# B&R Automation Studio project NewPendant_NG4_11_05_25A (part 10)

### HeadConfig.c
```c
/********************************************************************
 * COPYRIGHT --
 ********************************************************************
 * Package: FourAxisTigCtrl
 * File: HeadConfig.c
 * Author: ckaczkowski
 * Created: April 27, 2015
 * Directions - implemented 7 Febr 2018
   	TML_MTR_INST[i]._cfg.rev_motor - negative value change direction in Vel , Torq and Volt mode
	TML_MTR_INST[i]._cfg.rev_scale - negative value change pos and vel feedback (NOT Movement direction) and move direction in PT mode
 *******************************************************************/

#include <bur/plctypes.h>
#ifdef _DEFAULT_INCLUDES
	#include <AsDefault.h>
#endif

#include <math.h>

#ifndef _HEADCONFIG_C
#define _HEADCONFIG_C

#include <..\GlobDef.h>
#include <..\GlobDecl.h>
#include <..\..\Lib\LCDLib.c>

DINT NextDivider(DINT *in , DINT mod , BOOL dir);
DINT PickPinsNo(DINT *indx , DINT mod  );
void ParametrAssignToPointers(MASTER_typ *m  , UINT indx);

DINT ConfigureHead(MASTER_typ *m  , UINT headType );

DINT Configure_U_BEND_HP_PINS(MASTER_typ *m  , UINT headType );
DINT Configure_U_BEND_HP_ENC(MASTER_typ * m,UINT headType);
DINT Configure_OMEGA_16INCH_HP_ENCODER(MASTER_typ *m  , UINT headType );
DINT Configure_BPV_FACE_OSC(MASTER_typ * m, UINT headType);
DINT Configure_SUPER_MINI(MASTER_typ * m, UINT headType);
DINT Configure_U_BEND_HP_ENC_BEMF(MASTER_typ * m,UINT headType);
DINT Configure_BPV_F_HEAD(MASTER_typ * m, UINT headType);
DINT Configure_F_HEAD_HP_ENCODER(MASTER_typ * m,UINT headType);
DINT Configure_F_HEAD_HP_ENC_BEMF(MASTER_typ * m , UINT headType);
DINT Configure_BPV_FACE_OSC_ENC(MASTER_typ * m, UINT headType);
DINT Configure_BPV_FACE_OSC_EXP(MASTER_typ * m, UINT headType);
DINT Configure_BPV2_FACE_OSC_EXP(MASTER_typ * m, UINT headType);

DINT Configure_M_94(MASTER_typ * m, UINT headType);
DINT Configure_BPV_v2(MASTER_typ * m, UINT headType);
DINT Configure_MIG_TIG(MASTER_typ * m, UINT headType);

DINT Configure_BPV_v2_MPBO(MASTER_typ * m, UINT headType);
DINT Configure_BPV_v2_MPGH(MASTER_typ * m, UINT headType);
DINT Configure_BPV_v2_MPGV(MASTER_typ * m, UINT headType);

DINT Configure_BPV_v2_TT_BO(MASTER_typ * m, UINT headType);
DINT Configure_BPV_v2_MT_BO(MASTER_typ * m, UINT headType);

DINT Configure_BPV_v2_MT_BO_TOS(MASTER_typ * m, UINT headType);
DINT Configure_BPV_v2_TT_BO_TOS(MASTER_typ * m, UINT headType);

DINT  Configure_F_HEAD_HP_MINI_ENC(MASTER_typ * m,UINT headType);

DINT Configure_RUBIX(MASTER_typ * m, UINT headType);
DINT Configure_F_HEAD_MINI_STND(MASTER_typ * m,UINT headType);
DINT Configure_F_HEAD_MINI_OMEGA(MASTER_typ * m,UINT headType);
DINT Configure_D_HEAD_HP(MASTER_typ * m,UINT headType);

DINT Configure_CLAMSHELL_HEAD(MASTER_typ * m, UINT headType);
DINT Configure_CHERRYPOINT_BPV1_HEAD(MASTER_typ * m, UINT headType);
DINT Configure_CHERRYPOINT_BPV2_HEAD(MASTER_typ * m, UINT headType);
DINT Configure_CHERRYPOINT_MT_BP2_HEAD(MASTER_typ * m, UINT headType);

DINT  DefaultCalibr_U_BEND_HP_PINS(CurCalib_typ* defCalib);
DINT  DefaultCalibr_OMEGA_16INCH_HP_ENCODER(CurCalib_typ* defCalib);
DINT  DefaultCalibr_F_HEAD_HP_ENCODER(CurCalib_typ* defCalib);
DINT  DefaultCalibr_BPV_F_HEAD(CurCalib_typ* defCalib);

DINT Configure_BPV_v2_MT(MASTER_typ * m, UINT headType);
DINT Configure_BPV_V1_MT(MASTER_typ * m, UINT headType);

DINT  DefaultCalibr_F_HEAD_HP_MINI_ENC(CurCalib_typ* defCalib);
DINT  DefaultCalibr_U_BEND_HP_ENC(CurCalib_typ* defCalib);
DINT  DefaultCalibr_BPV_FACE_OSC(CurCalib_typ* defCalib);
DINT  DefaultCalibr_SUPER_MINI(CurCalib_typ* defCalib);
DINT  DefaultCalibr_U_BEND_HP_ENC_BEMF(CurCalib_typ* defCalib);
DINT  DefaultCalibr_F_HEAD_HP_ENC_BEMF(CurCalib_typ* defCalib);
DINT  DefaultCalibr_M_94(CurCalib_typ* defCalib);
DINT  DefaultCalibr_BPV_v2(CurCalib_typ* defCalib);
DINT  DefaultCalibr_BPV_v2_MPBO(CurCalib_typ* defCalib);
DINT  DefaultCalibr_BPV_v2_MPGH(CurCalib_typ* defCalib);
DINT  DefaultCalibr_BPV_v2_MPGV(CurCalib_typ* defCalib);

DINT  DefaultCalibr_BPV_v2_TT_BO(CurCalib_typ* defCalib);
DINT  DefaultCalibr_BPV_v2_MT_BO(CurCalib_typ* defCalib);

DINT  DefaultCalibr_BPV_v2_MT_BO_TOS(CurCalib_typ* defCalib);
DINT  DefaultCalibr_BPV_v2_TT_BO_TOS(CurCalib_typ* defCalib);

DINT  DefaultCalibr_RUBIX(CurCalib_typ* defCalib);
DINT  DefaultCalibr_F_HEAD_MINI_STND(CurCalib_typ* defCalib);
DINT  DefaultCalibr_F_HEAD_MINI_OMEGA(CurCalib_typ* defCalib);
DINT  DefaultCalibr_D_HEAD_HP(CurCalib_typ* defCalib);

DINT  DefaultCalibr_BPV_v2_MT(CurCalib_typ* defCalib);
DINT  DefaultCalibr_BPV_V1_MT(CurCalib_typ* defCalib);

DINT  DefaultCalibr_CLAMSHELL_HEAD(CurCalib_typ* defCalib);
DINT  DefaultCalibr_CHERRYPOINT_BPV1_HEAD(CurCalib_typ* defCalib);
DINT  DefaultCalibr_CHERRYPOINT_BPV2_HEAD(CurCalib_typ* defCalib);
DINT  DefaultCalibr_MIG_TIG(CurCalib_typ* defCalib);

float Gen_one;

DINT ConfigureHead(MASTER_typ *m  , UINT headType ){
int i;

CurCfg_typ *curCfg;
Cfg_typ *cfg;
CurCalib_typ *curCalib , *defaultCalib;

	if(!m)
		return;

	curCfg = (CurCfg_typ*)m->pCurCfg;
	cfg = (Cfg_typ*)m->pCfg;

	curCalib = m->pCalib;
	defaultCalib = m->pDefaultCalib;

	if(!curCfg || !cfg || !curCalib  || !defaultCalib)
		return;

	///
	if(curCalib->GenSetup[SETUP_POLE_ELEMENTS] < 2)
		curCalib->GenSetup[SETUP_POLE_ELEMENTS] = 2;

	else if(curCalib->GenSetup[SETUP_POLE_ELEMENTS] > 32)
		curCalib->GenSetup[SETUP_POLE_ELEMENTS] = 32;
	/////////

	for(i = 0 ; i < PROCESS_NUM ; i++)
		Process[i].ConfigReady = 0;

	for(i = 0 ; i < TML_SERVO_NUM ; i++){
		TML_MTR_INST[i].pState = 0;
		TML_MTR_INST[i]._cfg.NotAutoDownload = 0; // Default - auto download setup
		TML_MTR_INST[i]._cfg.MtrType = 0; // Default - DC Motor
	}

	for(i=0 ; i < VECTORS_NUM; i++){

		VectorStateMach[i].Indx = i;
	}

	// This is only to not forget Synch Configuration
	WIRE_Param_Set[0].pSynchMode = &WFSynchMode;
	WIRE_Param_Set[0].pSynchClock = &SynchClckToWF;

	WIRE_Param_Set[1].pSynchMode = &WPSynchMode;
	WIRE_Param_Set[1].pSynchClock = &SynchClckToWP;

	TVL_ROT_Param_Set[0].pSynchMode = &TVLSynchMode;
	TVL_ROT_Param_Set[0].pSynchClock = &SynchClckToTVL;

	////////////   NEW HEAD Configuration - will be from file parser   /////////////////////
	switch(headType){
		/************ 0 **********/
		case U_BEND_HP_PINS:

			// TVL
			m->pCfg->HeadCfg.SwitchHead.VECT_Indx = 0;
			m->pCfg->HeadCfg.SwitchHead.TML_Indx = 0;

			m->pCfg->HeadCfg.TVL.PROC_Indx = PROC_TVL;
			m->pCfg->HeadCfg.TVL.TML_Indx = TML_AX_TVL;
			m->pCfg->HeadCfg.TVL.DC_Indx = 0;

			m->pCfg->HeadCfg.TVL.VECT_Indx = VECT_TVL;
			m->pCfg->HeadCfg.TVL.Enc_Dir = 1;
			m->pCfg->HeadCfg.TVL.EncPerTick = 160;
			m->pCfg->HeadCfg.TVL.PinsPerRot = 0;  // Dynamic Configuration
			m->pCfg->HeadCfg.TVL.DistPerTick = 25.4 / 4.0; // 1/4"

			// Lamp On Off
			m->pCfg->HeadCfg.LampOnOFF.VECT_A_Indx = 0; // 0 - not used
			m->pCfg->HeadCfg.LampOnOFF.VECT_B_Indx = 0; // 0 - not used

			// INDX
			m->pCfg->HeadCfg.INDX.PROC_Indx = PROC_INDX; // Must be even is disabled

			m->pCfg->HeadCfg.OSC.DwellDir = 1;

		break;

		/************ 1 ************/
		case U_BEND_HP_ENC:

			m->pCfg->HeadCfg.GEN.Torch_Mode = MODE_SINGLE_TORCH;

			// TVL
			m->pCfg->HeadCfg.SwitchHead.VECT_Indx = 0;
			m->pCfg->HeadCfg.SwitchHead.TML_Indx = 0;

			m->pCfg->HeadCfg.TVL.PROC_Indx = PROC_TVL;
			m->pCfg->HeadCfg.TVL.TML_Indx = TML_AX_TVL;
			m->pCfg->HeadCfg.TVL.DC_Indx = 0;

			m->pCfg->HeadCfg.TVL.VECT_Indx = VECT_TVL;
			m->pCfg->HeadCfg.TVL.Enc_Dir = 1;
			m->pCfg->HeadCfg.TVL.EncPerTick = 200; // (4000 * 4) / (10 * 1/4") * 32 ( becaue 1/32" is one tick")
			m->pCfg->HeadCfg.TVL.PinsPerRot = 640;  // 80 pins , 1/4" per pin
			m->pCfg->HeadCfg.TVL.DistPerTick = 25.4 /32.0; // 1/32"

			m->pCfg->HeadCfg.TVL.BtnJog_Gain = 24;
			m->pCfg->HeadCfg.TVL.BtnJog_Mode = BTN_JOG_MODE_SINGLE;

			// WF
			m->pCfg->HeadCfg.WF.PROC_Indx = PROC_WIRE_FEED;
			m->pCfg->HeadCfg.WF.VECT_A_Indx = VECT_WF;
			m->pCfg->HeadCfg.WF.VECT_B_Indx = VECT_WF_1;
			m->pCfg->HeadCfg.WF.DC_A_Indx = DC_AX_WF;
			m->pCfg->HeadCfg.WF.DC_B_Indx = DC_AX_WF_1;

			m->pCfg->HeadCfg.WF.BtnJog_Gain = 24;
			m->pCfg->HeadCfg.WF.BtnJog_Mode = BTN_JOG_MODE_SINGLE;

			// WP
			m->pCfg->HeadCfg.WP.PROC_Indx = PROC_WIRE_PULSE;
			m->pCfg->HeadCfg.WP.VECT_A_Indx = VECT_WP;
			m->pCfg->HeadCfg.WP.VECT_B_Indx = VECT_WP_1;
			m->pCfg->HeadCfg.WP.DC_A_Indx = DC_AX_WP;
			m->pCfg->HeadCfg.WP.DC_B_Indx = DC_AX_WP_1;

			// OSC
			m->pCfg->HeadCfg.OSC.PROC_Indx = PROC_OSC;
			m->pCfg->HeadCfg.OSC.VECT_A_Indx = VECT_OSC;
			m->pCfg->HeadCfg.OSC.VECT_B_Indx = VECT_OSC;
			m->pCfg->HeadCfg.OSC.TML_A_Indx = TML_AX_OSC;
			m->pCfg->HeadCfg.OSC.TML_B_Indx = TML_AX_OSC;
			m->pCfg->HeadCfg.OSC.Limits_Harcoded = 0;

			m->pCfg->HeadCfg.OSC.BtnJog_Gain = 24.0;
			m->pCfg->HeadCfg.OSC.BtnJog_Mode = BTN_JOG_MODE_SINGLE;

			m->pCfg->HeadCfg.OSC.WheelJog_Gain1 = 5;
			m->pCfg->HeadCfg.OSC.WhelJog_Mode1 = WHL_JOG_MODE_STEP;

			m->pCfg->HeadCfg.OSC.WheelJog_Gain2 = 0.2;
			m->pCfg->HeadCfg.OSC.WhelJog_Mode2 = WHL_JOG_MODE_STEP;
			m->pCfg->HeadCfg.OSC.WhelJog_OnlyWhenRun = 1;

			m->pCfg->HeadCfg.OSC.DwellDir = 1;

			// AVC
			m->pCfg->HeadCfg.AVC.PROC_Indx = PROC_AVC;
			m->pCfg->HeadCfg.AVC.VECT_A_Indx = VECT_AVC;
			m->pCfg->HeadCfg.AVC.VECT_B_Indx = VECT_AVC;
			m->pCfg->HeadCfg.AVC.TML_A_Indx = TML_AX_AVC;
			m->pCfg->HeadCfg.AVC.TML_B_Indx = TML_AX_AVC;

			m->pCfg->HeadCfg.AVC.BtnJog_Gain = 24;
			m->pCfg->HeadCfg.AVC.BtnJog_Mode = BTN_JOG_MODE_SINGLE;

			// GAS
			m->pCfg->HeadCfg.GAS.PROC_Indx = PROC_GAS;

			// COOL
			m->pCfg->HeadCfg.COOL.PROC_Indx = PROC_COOL;

			// TIG
			m->pCfg->HeadCfg.TIG.PROC_Indx = PROC_TIG_PS;

			// HW
			m->pCfg->HeadCfg.HW.PROC_Indx = PROC_HW_PS;

			// INDX
			m->pCfg->HeadCfg.INDX.PROC_Indx = PROC_INDX; // Must be even is disabled

			// WB
			m->pCfg->HeadCfg.WB[WB_UD].PROC_Indx = PROC_WB_UD;
			m->pCfg->HeadCfg.WB[WB_LR].PROC_Indx = PROC_WB_LR;

			m->pCfg->HeadCfg.WB[WB_UD].VECT_Indx = VECT_WB_UD;
			m->pCfg->HeadCfg.WB[WB_LR].VECT_Indx = VECT_WB_LR;

			// Lamp On Off
			m->pCfg->HeadCfg.LampOnOFF.VECT_A_Indx = 0; // 0 - not used
			m->pCfg->HeadCfg.LampOnOFF.VECT_B_Indx = 0; // 0 - not used

			// frame size if zero always speed factor is 1.0
			m->FrameDia = 4.5 * in_2_mm ;
			m->FrameDia = 0.0;

			Configure_U_BEND_HP_ENC(m , U_BEND_HP_ENC);
			DefaultCalibr_U_BEND_HP_ENC(m->pDefaultCalib);

		break;

		/************ 2 ************/
		case F_HEAD_HP_ENCODER:

			m->pCfg->HeadCfg.GEN.Torch_Mode = MODE_SINGLE_TORCH;

			// TVL
			m->pCfg->HeadCfg.SwitchHead.VECT_Indx = 0;
			m->pCfg->HeadCfg.SwitchHead.TML_Indx = 0;

			m->pCfg->HeadCfg.TVL.PROC_Indx = PROC_TVL;
			m->pCfg->HeadCfg.TVL.TML_Indx = TML_AX_TVL;
			m->pCfg->HeadCfg.TVL.DC_Indx = 0;

			m->pCfg->HeadCfg.TVL.VECT_Indx = VECT_TVL;
			m->pCfg->HeadCfg.TVL.Enc_Dir = 1;
			m->pCfg->HeadCfg.TVL.EncPerTick = 38;  // 1/16 inch
			m->pCfg->HeadCfg.TVL.PinsPerRot = 0;  // Dynamic Configuration
			m->pCfg->HeadCfg.TVL.DistPerTick = 25.4 /16.0; // 1/16"

			m->pCfg->HeadCfg.TVL.BtnJog_Gain = 24;
			m->pCfg->HeadCfg.TVL.BtnJog_Mode = BTN_JOG_MODE_SINGLE;

			// WF
			m->pCfg->HeadCfg.WF.PROC_Indx = PROC_WIRE_FEED;
			m->pCfg->HeadCfg.WF.VECT_A_Indx = VECT_WF;
			m->pCfg->HeadCfg.WF.VECT_B_Indx = VECT_WF_1;
			m->pCfg->HeadCfg.WF.DC_A_Indx = DC_AX_WF;
			m->pCfg->HeadCfg.WF.DC_B_Indx = DC_AX_WF_1;

			m->pCfg->HeadCfg.WF.BtnJog_Gain = 24;
			m->pCfg->HeadCfg.WF.BtnJog_Mode = BTN_JOG_MODE_SINGLE;

			// WP
			m->pCfg->HeadCfg.WP.PROC_Indx = PROC_WIRE_PULSE;
			m->pCfg->HeadCfg.WP.VECT_A_Indx = VECT_WP;
			m->pCfg->HeadCfg.WP.VECT_B_Indx = VECT_WP_1;
			m->pCfg->HeadCfg.WP.DC_A_Indx = DC_AX_WP;
			m->pCfg->HeadCfg.WP.DC_B_Indx = DC_AX_WP_1;

			// OSC
			m->pCfg->HeadCfg.OSC.PROC_Indx = PROC_OSC;
			m->pCfg->HeadCfg.OSC.VECT_A_Indx = VECT_OSC;
			m->pCfg->HeadCfg.OSC.VECT_B_Indx = VECT_OSC;
			m->pCfg->HeadCfg.OSC.TML_A_Indx = TML_AX_OSC;
			m->pCfg->HeadCfg.OSC.TML_B_Indx = TML_AX_OSC;
			m->pCfg->HeadCfg.OSC.Limits_Harcoded = 0;

			m->pCfg->HeadCfg.OSC.BtnJog_Gain = 24.0;
			m->pCfg->HeadCfg.OSC.BtnJog_Mode = BTN_JOG_MODE_SINGLE;

			m->pCfg->HeadCfg.OSC.WheelJog_Gain1 = 5.0;
			m->pCfg->HeadCfg.OSC.WhelJog_Mode1 = WHL_JOG_MODE_STEP;

			m->pCfg->HeadCfg.OSC.WheelJog_Gain2 = 0.2;
			m->pCfg->HeadCfg.OSC.WhelJog_Mode2 = WHL_JOG_MODE_STEP;
			m->pCfg->HeadCfg.OSC.WhelJog_OnlyWhenRun = 1;

			m->pCfg->HeadCfg.OSC.DwellDir = 1;

			// AVC
			m->pCfg->HeadCfg.AVC.PROC_Indx = PROC_AVC;
			m->pCfg->HeadCfg.AVC.VECT_A_Indx = VECT_AVC;
			m->pCfg->HeadCfg.AVC.VECT_B_Indx = VECT_AVC;
			m->pCfg->HeadCfg.AVC.TML_A_Indx = TML_AX_AVC;
			m->pCfg->HeadCfg.AVC.TML_B_Indx = TML_AX_AVC;

			m->pCfg->HeadCfg.AVC.BtnJog_Gain = 24;
			m->pCfg->HeadCfg.AVC.BtnJog_Mode = BTN_JOG_MODE_SINGLE;

			// GAS
			m->pCfg->HeadCfg.GAS.PROC_Indx = PROC_GAS;

			// COOL
			m->pCfg->HeadCfg.COOL.PROC_Indx = PROC_COOL;

			// TIG
			m->pCfg->HeadCfg.TIG.PROC_Indx = PROC_TIG_PS;

			// HW
			m->pCfg->HeadCfg.HW.PROC_Indx = PROC_HW_PS;

			// INDX
			m->pCfg->HeadCfg.INDX.PROC_Indx = PROC_INDX; // Must be even is disabled

			// WB
			m->pCfg->HeadCfg.WB[WB_UD].PROC_Indx = PROC_WB_UD;
			m->pCfg->HeadCfg.WB[WB_LR].PROC_Indx = PROC_WB_LR;

			m->pCfg->HeadCfg.WB[WB_UD].VECT_Indx = VECT_WB_UD;
			m->pCfg->HeadCfg.WB[WB_LR].VECT_Indx = VECT_WB_LR;

			// Lamp On Off
			m->pCfg->HeadCfg.LampOnOFF.VECT_A_Indx = 0; // 0 - not used
			m->pCfg->HeadCfg.LampOnOFF.VECT_B_Indx = 0; // 0 - not used

			/////////////////////////////////////////////////////

			// frame size if zero always speed factor is 1.0
			//m->FrameDia = 4.5 * in_2_mm ;
			m->FrameDia = 0.0;

			Configure_F_HEAD_HP_ENCODER(m , F_HEAD_HP_ENCODER);
			DefaultCalibr_F_HEAD_HP_ENCODER(m->pDefaultCalib);

		break;

		/************ 3 ************/
		/************ 29 ************/
		case BPV_F_HEAD:
		case BPV_v1_MT:

			m->pCfg->HeadCfg.GEN.Torch_Mode = MODE_SINGLE_TORCH;

			// TVL
			m->pCfg->HeadCfg.SwitchHead.VECT_Indx = 0;
			m->pCfg->HeadCfg.SwitchHead.TML_Indx = 0;

			m->pCfg->HeadCfg.TVL.PROC_Indx = PROC_TVL;
			m->pCfg->HeadCfg.TVL.TML_Indx = TML_AX_TVL;

			m->pCfg->HeadCfg.TVL.VECT_Indx = VECT_TVL;
			m->pCfg->HeadCfg.TVL.Enc_Dir = 1;
			//m->pCfg->HeadCfg.TVL.EncPerTick  = 5085;  //  5084.8094458543457034129135792358	// For 1/32 "
			m->pCfg->HeadCfg.TVL.EncPerTick  = 5088; // aby bylo 32 razy
			m->pCfg->HeadCfg.TVL.EncPerTick_SecEnc = 159; // (4000 * 4) / (1" * Pi * 32)
			m->pCfg->HeadCfg.TVL.PinsPerRot = 0;  // Dynamic Configuration
			m->pCfg->HeadCfg.TVL.DistPerTick = 25.4 /32.0; // 1/32"

			m->pCfg->HeadCfg.TVL.BtnJog_Gain = 24;
			m->pCfg->HeadCfg.TVL.BtnJog_Mode = BTN_JOG_MODE_SINGLE;

			// WF
			m->pCfg->HeadCfg.WF.PROC_Indx = PROC_WIRE_FEED;
			m->pCfg->HeadCfg.WF.VECT_A_Indx = VECT_WF;
			m->pCfg->HeadCfg.WF.VECT_B_Indx = VECT_WF_1;
			m->pCfg->HeadCfg.WF.TML_A_Indx = TML_AX_WF;
			m->pCfg->HeadCfg.WF.TML_B_Indx = TML_AX_WF_1;

			m->pCfg->HeadCfg.WF.BtnJog_Gain = 24;
			m->pCfg->HeadCfg.WF.BtnJog_Mode = BTN_JOG_MODE_SINGLE;

			// WP
			m->pCfg->HeadCfg.WP.PROC_Indx = PROC_WIRE_PULSE;
			m->pCfg->HeadCfg.WP.VECT_A_Indx = VECT_WP;
			m->pCfg->HeadCfg.WP.VECT_B_Indx = VECT_WP_1;
			m->pCfg->HeadCfg.WP.TML_A_Indx = TML_AX_WP;
			m->pCfg->HeadCfg.WP.TML_B_Indx = TML_AX_WP_1;

			// OSC
			m->pCfg->HeadCfg.OSC.PROC_Indx = PROC_OSC;
			m->pCfg->HeadCfg.OSC.VECT_A_Indx = VECT_OSC;
			m->pCfg->HeadCfg.OSC.VECT_B_Indx = VECT_OSC;
			m->pCfg->HeadCfg.OSC.TML_A_Indx = TML_AX_OSC;
			m->pCfg->HeadCfg.OSC.TML_B_Indx = TML_AX_OSC;
			m->pCfg->HeadCfg.OSC.Limits_Harcoded = 0;

			m->pCfg->HeadCfg.OSC.WhelJog_OnlyWhenRun = 0;

			m->pCfg->HeadCfg.OSC.BtnJog_Gain = 4;
			m->pCfg->HeadCfg.OSC.BtnJog_Mode = BTN_JOG_MODE_SINGLE;

			m->pCfg->HeadCfg.OSC.WheelJog_Gain1 = 0.2;
			m->pCfg->HeadCfg.OSC.WhelJog_Mode1 = WHL_JOG_MODE_STEP;

			m->pCfg->HeadCfg.OSC.WheelJog_Gain2 = 0.2;
			m->pCfg->HeadCfg.OSC.WhelJog_Mode2 = WHL_JOG_MODE_STEP;

			m->pCfg->HeadCfg.OSC.DwellDir = 1;

			// WRST
			m->pCfg->HeadCfg.WRST.PROC_Indx = PROC_WRST;
			m->pCfg->HeadCfg.WRST.VECT_A_Indx = VECT_WRST;
			m->pCfg->HeadCfg.WRST.VECT_B_Indx = VECT_WRST;
			m->pCfg->HeadCfg.WRST.TML_A_Indx = TML_AX_WRST;
			m->pCfg->HeadCfg.WRST.TML_B_Indx = TML_AX_WRST;
			m->pCfg->HeadCfg.WRST.Limits_Harcoded = 0;

			m->pCfg->HeadCfg.WRST.BtnJog_Gain = 24.0;
			m->pCfg->HeadCfg.WRST.BtnJog_Mode = BTN_JOG_MODE_SINGLE;

			// AVC
			m->pCfg->HeadCfg.AVC.PROC_Indx = PROC_AVC;
			m->pCfg->HeadCfg.AVC.VECT_A_Indx = VECT_AVC;
			m->pCfg->HeadCfg.AVC.VECT_B_Indx = VECT_AVC;
			m->pCfg->HeadCfg.AVC.TML_A_Indx = TML_AX_AVC;
			m->pCfg->HeadCfg.AVC.TML_B_Indx = TML_AX_AVC;

			m->pCfg->HeadCfg.AVC.BtnJog_Gain = 1;
			m->pCfg->HeadCfg.AVC.BtnJog_Mode = BTN_JOG_MODE_SINGLE;

			// GAS
			m->pCfg->HeadCfg.GAS.PROC_Indx = PROC_GAS;

			// COOL
			m->pCfg->HeadCfg.COOL.PROC_Indx = PROC_COOL;

			// TIG
			m->pCfg->HeadCfg.TIG.PROC_Indx = PROC_TIG_PS;

			// HW
			m->pCfg->HeadCfg.HW.PROC_Indx = PROC_HW_PS;

			// INDX
			m->pCfg->HeadCfg.INDX.PROC_Indx = PROC_INDX;
			m->pCfg->HeadCfg.INDX.VECT_A_Indx = VECT_INDX_1;
			m->pCfg->HeadCfg.INDX.VECT_B_Indx = VECT_INDX_2;
			m->pCfg->HeadCfg.INDX.DC_A_Indx = DC_INDX_1;
			m->pCfg->HeadCfg.INDX.DC_B_Indx = DC_INDX_2;
			m->pCfg->HeadCfg.INDX.BtnJog_Gain = 1.0;

			// WB
			m->pCfg->HeadCfg.WB[WB_UD].PROC_Indx = PROC_WB_UD;
			m->pCfg->HeadCfg.WB[WB_LR].PROC_Indx = PROC_WB_LR;

			m->pCfg->HeadCfg.WB[WB_UD].VECT_Indx = VECT_WB_UD;
			m->pCfg->HeadCfg.WB[WB_LR].VECT_Indx = VECT_WB_LR;

			// Lamp On Off
			m->pCfg->HeadCfg.LampOnOFF.VECT_A_Indx = 0; // 0 - not used
			m->pCfg->HeadCfg.LampOnOFF.VECT_B_Indx = 0; // 0 - not used

			/////////////////////////////////////////////////////

			// frame size if zero always speed factor is 1.0
			//m->FrameDia = 4.5 * in_2_mm ;
			m->FrameDia = 0.0;

			switch(headType){

				case BPV_F_HEAD:
					Configure_BPV_F_HEAD(m , BPV_F_HEAD);
					DefaultCalibr_BPV_F_HEAD(m->pDefaultCalib);
				break;

				case BPV_v1_MT:
					Configure_BPV_V1_MT(m , BPV_v1_MT);
					DefaultCalibr_BPV_V1_MT(m->pDefaultCalib);
				break;
			}

		break;

		/************ 4 ************/
		case OMEGA_16INCH_HP_ENCODER:

			// TVL
			m->pCfg->HeadCfg.SwitchHead.VECT_Indx = 0;
			m->pCfg->HeadCfg.SwitchHead.TML_Indx = 0;

			m->pCfg->HeadCfg.TVL.PROC_Indx = PROC_TVL;
			m->pCfg->HeadCfg.TVL.TML_Indx = TML_AX_TVL;
			m->pCfg->HeadCfg.TVL.DC_Indx = 0;

			m->pCfg->HeadCfg.TVL.VECT_Indx = VECT_TVL;
			m->pCfg->HeadCfg.TVL.Enc_Dir = 1;
			m->pCfg->HeadCfg.TVL.PinsPerRot  = 1024;
			m->pCfg->HeadCfg.TVL.EncPerTick = 10312656 * 4 / m->pCfg->HeadCfg.TVL.PinsPerRot  ;
			curCalib->GenSetup[SETUP_PIN_PER_ROT] = m->pCfg->HeadCfg.TVL.PinsPerRot;
			m->pCfg->HeadCfg.TVL.DistPerTick = 25.4 /16.0; // ????????????????????????

			// INDX
			m->pCfg->HeadCfg.INDX.PROC_Indx = PROC_INDX; // Must be even is disabled

			// Lamp On Off
			m->pCfg->HeadCfg.LampOnOFF.VECT_A_Indx = 0; // 0 - not used
			m->pCfg->HeadCfg.LampOnOFF.VECT_B_Indx = 0; // 0 - not used

		break;

		/************ 5 ************/
		case OMEGA_10INCH_HP_ENCODER:

			// TVL
			m->pCfg->HeadCfg.SwitchHead.VECT_Indx = 0;
			m->pCfg->HeadCfg.SwitchHead.TML_Indx = 0;

			m->pCfg->HeadCfg.TVL.PROC_Indx = PROC_TVL;
			m->pCfg->HeadCfg.TVL.TML_Indx = TML_AX_TVL;
			m->pCfg->HeadCfg.TVL.DC_Indx = 0;

			m->pCfg->HeadCfg.TVL.VECT_Indx = VECT_TVL;
			m->pCfg->HeadCfg.TVL.Enc_Dir = 1;
			m->pCfg->HeadCfg.TVL.PinsPerRot  = 1024;
			m->pCfg->HeadCfg.TVL.EncPerTick = 10312656 * 4 / m->pCfg->HeadCfg.TVL.PinsPerRot  ;
			curCalib->GenSetup[SETUP_PIN_PER_ROT] = m->pCfg->HeadCfg.TVL.PinsPerRot;
			m->pCfg->HeadCfg.TVL.DistPerTick = 25.4 /16.0; // ????????????????????????

			// INDX
			m->pCfg->HeadCfg.INDX.PROC_Indx = PROC_INDX; // Must be even is disabled

			// Lamp On Off
			m->pCfg->HeadCfg.LampOnOFF.VECT_A_Indx = 0; // 0 - not used
			m->pCfg->HeadCfg.LampOnOFF.VECT_B_Indx = 0; // 0 - not used

		break;

		/************ 6 ************/
		case OMEGA_8INCH_HP_ENCODER:

			// TVL
			m->pCfg->HeadCfg.SwitchHead.VECT_Indx = 0;
			m->pCfg->HeadCfg.SwitchHead.TML_Indx = 0;

			m->pCfg->HeadCfg.TVL.PROC_Indx = PROC_TVL;
			m->pCfg->HeadCfg.TVL.TML_Indx = TML_AX_TVL;
			m->pCfg->HeadCfg.TVL.DC_Indx = 0;

			m->pCfg->HeadCfg.TVL.VECT_Indx = VECT_TVL;
			m->pCfg->HeadCfg.TVL.Enc_Dir = 1;
			m->pCfg->HeadCfg.TVL.PinsPerRot  = 1024;
			m->pCfg->HeadCfg.TVL.EncPerTick = 10312656 * 4 / m->pCfg->HeadCfg.TVL.PinsPerRot  ;
			curCalib->GenSetup[SETUP_PIN_PER_ROT] = m->pCfg->HeadCfg.TVL.PinsPerRot;
			m->pCfg->HeadCfg.TVL.DistPerTick = 25.4 /16.0; // ????????????????????????

			// INDX
			m->pCfg->HeadCfg.INDX.PROC_Indx = PROC_INDX; // Must be even is disabled

			// Lamp On Off
			m->pCfg->HeadCfg.LampOnOFF.VECT_A_Indx = 0; // 0 - not used
			m->pCfg->HeadCfg.LampOnOFF.VECT_B_Indx = 0; // 0 - not used

		break;

		/************ 7 ************/
		case F_HEAD_HP_MINI_ENC:

			m->pCfg->HeadCfg.GEN.Torch_Mode = MODE_SINGLE_TORCH;

			// TVL
			m->pCfg->HeadCfg.SwitchHead.VECT_Indx = 0;
			m->pCfg->HeadCfg.SwitchHead.TML_Indx = 0;

			m->pCfg->HeadCfg.TVL.PROC_Indx = PROC_TVL;
			m->pCfg->HeadCfg.TVL.TML_Indx = TML_AX_TVL;
			m->pCfg->HeadCfg.TVL.DC_Indx = 0;

			m->pCfg->HeadCfg.TVL.VECT_Indx = VECT_TVL;
			m->pCfg->HeadCfg.TVL.Enc_Dir = 1;
			m->pCfg->HeadCfg.TVL.EncPerTick = 38;  // 1/16 inch
			m->pCfg->HeadCfg.TVL.PinsPerRot = 0;  // Dynamic Configuration
			m->pCfg->HeadCfg.TVL.DistPerTick = 25.4 /16.0; // 1/16"

			m->pCfg->HeadCfg.TVL.BtnJog_Gain = 24;
			m->pCfg->HeadCfg.TVL.BtnJog_Mode = BTN_JOG_MODE_SINGLE;

			// WF
			m->pCfg->HeadCfg.WF.PROC_Indx = PROC_WIRE_FEED;
			m->pCfg->HeadCfg.WF.VECT_A_Indx = VECT_WF;
			m->pCfg->HeadCfg.WF.VECT_B_Indx = VECT_WF;
			m->pCfg->HeadCfg.WF.DC_A_Indx = DC_AX_WF;
			m->pCfg->HeadCfg.WF.DC_B_Indx = DC_AX_WF;

			m->pCfg->HeadCfg.WF.BtnJog_Gain = 24;
			m->pCfg->HeadCfg.WF.BtnJog_Mode = BTN_JOG_MODE_SINGLE;

			// WP
			m->pCfg->HeadCfg.WP.PROC_Indx = PROC_WIRE_PULSE;
			m->pCfg->HeadCfg.WP.VECT_A_Indx = VECT_WP;
			m->pCfg->HeadCfg.WP.VECT_B_Indx = VECT_WP;
			m->pCfg->HeadCfg.WP.DC_A_Indx = DC_AX_WP;
			m->pCfg->HeadCfg.WP.DC_B_Indx = DC_AX_WP;

			// OSC
			m->pCfg->HeadCfg.OSC.PROC_Indx = PROC_OSC;
			m->pCfg->HeadCfg.OSC.VECT_A_Indx = VECT_OSC;
			m->pCfg->HeadCfg.OSC.VECT_B_Indx = VECT_OSC;
			m->pCfg->HeadCfg.OSC.TML_A_Indx = TML_AX_OSC;
			m->pCfg->HeadCfg.OSC.TML_B_Indx = TML_AX_OSC;
			m->pCfg->HeadCfg.OSC.Limits_Harcoded = 0;

			m->pCfg->HeadCfg.OSC.BtnJog_Gain = 24.0;
			m->pCfg->HeadCfg.OSC.BtnJog_Mode = BTN_JOG_MODE_SINGLE;

			m->pCfg->HeadCfg.OSC.WheelJog_Gain1 = 5;
			m->pCfg->HeadCfg.OSC.WhelJog_Mode1 = WHL_JOG_MODE_STEP;

			m->pCfg->HeadCfg.OSC.WheelJog_Gain2 = 0.2;
			m->pCfg->HeadCfg.OSC.WhelJog_Mode2 = WHL_JOG_MODE_STEP;
			m->pCfg->HeadCfg.OSC.WhelJog_OnlyWhenRun = 1;

			m->pCfg->HeadCfg.OSC.DwellDir = 1;

			// AVC
			m->pCfg->HeadCfg.AVC.PROC_Indx = PROC_AVC;
			m->pCfg->HeadCfg.AVC.VECT_A_Indx = VECT_AVC;
			m->pCfg->HeadCfg.AVC.VECT_B_Indx = VECT_AVC;
			m->pCfg->HeadCfg.AVC.TML_A_Indx = TML_AX_AVC;
			m->pCfg->HeadCfg.AVC.TML_B_Indx = TML_AX_AVC;

			m->pCfg->HeadCfg.AVC.BtnJog_Gain = 24;
			m->pCfg->HeadCfg.AVC.BtnJog_Mode = BTN_JOG_MODE_SINGLE;

			// GAS
			m->pCfg->HeadCfg.GAS.PROC_Indx = PROC_GAS;

			// COOL
			m->pCfg->HeadCfg.COOL.PROC_Indx = PROC_COOL;

			// TIG
			m->pCfg->HeadCfg.TIG.PROC_Indx = PROC_TIG_PS;

			// HW
			m->pCfg->HeadCfg.HW.PROC_Indx = PROC_HW_PS;

			// INDX
			m->pCfg->HeadCfg.INDX.PROC_Indx = PROC_INDX; // Must be even is disabled

			// WB
			m->pCfg->HeadCfg.WB[WB_UD].PROC_Indx = PROC_WB_UD;
			m->pCfg->HeadCfg.WB[WB_LR].PROC_Indx = PROC_WB_LR;

			m->pCfg->HeadCfg.WB[WB_UD].VECT_Indx = VECT_WB_UD;
			m->pCfg->HeadCfg.WB[WB_LR].VECT_Indx = VECT_WB_LR;

			// Lamp On Off
			m->pCfg->HeadCfg.LampOnOFF.VECT_A_Indx = 0; // 0 - not used
			m->pCfg->HeadCfg.LampOnOFF.VECT_B_Indx = 0; // 0 - not used

			//////////////////////
			// frame size if zero always speed factor is 1.0
			//m->FrameDia = 4.5 * in_2_mm ;
			m->FrameDia = 0.0;

			Configure_F_HEAD_HP_MINI_ENC(m , F_HEAD_HP_MINI_ENC);
			DefaultCalibr_F_HEAD_HP_MINI_ENC(m->pDefaultCalib);

		break;

		/************ SUPER_MINI - 8 ************/
		case SUPER_MINI:

			m->pCfg->HeadCfg.GEN.Torch_Mode = MODE_SINGLE_TORCH;

			// TVL
			m->pCfg->HeadCfg.SwitchHead.VECT_Indx = VECT_TVL+1;
			m->pCfg->HeadCfg.SwitchHead.TML_Indx = TML_AX_TVL+1;

			m->pCfg->HeadCfg.TVL.PROC_Indx = PROC_TVL;
			m->pCfg->HeadCfg.TVL.TML_Indx = TML_AX_TVL;

			m->pCfg->HeadCfg.TVL.VECT_Indx = VECT_TVL;
			m->pCfg->HeadCfg.TVL.Enc_Dir = -1;
			m->pCfg->HeadCfg.TVL.EncPerTick  = (1024 * 4 * (300564/1300) * (36.0/33.0)) / (1.25 * M_PI * 32); //5088;
			m->pCfg->HeadCfg.TVL.EncPerTick_SecEnc = 255; // (4000 * 4) / (0.625 * Pi * 32)
			m->pCfg->HeadCfg.TVL.PinsPerRot = 0;  // Dynamic Configuration
			m->pCfg->HeadCfg.TVL.DistPerTick = 25.4 /32.0; // 1/32"

			m->pCfg->HeadCfg.TVL.BtnJog_Gain = 24;
			m->pCfg->HeadCfg.TVL.BtnJog_Mode = BTN_JOG_MODE_SINGLE;

			// WF
			m->pCfg->HeadCfg.WF.PROC_Indx = PROC_WIRE_FEED;
			m->pCfg->HeadCfg.WF.VECT_A_Indx = VECT_WF;
			m->pCfg->HeadCfg.WF.VECT_B_Indx = VECT_WF;
			m->pCfg->HeadCfg.WF.TML_A_Indx = TML_AX_WF;
			m->pCfg->HeadCfg.WF.TML_B_Indx = TML_AX_WF;

			m->pCfg->HeadCfg.WF.BtnJog_Gain = 24;
			m->pCfg->HeadCfg.WF.BtnJog_Mode = BTN_JOG_MODE_SINGLE;

			// WP
			m->pCfg->HeadCfg.WP.PROC_Indx = PROC_WIRE_PULSE;
			m->pCfg->HeadCfg.WP.VECT_A_Indx = VECT_WP;
			m->pCfg->HeadCfg.WP.VECT_B_Indx = VECT_WP;
			m->pCfg->HeadCfg.WP.TML_A_Indx = TML_AX_WP;
			m->pCfg->HeadCfg.WP.TML_B_Indx = TML_AX_WP;

			// OSC
			m->pCfg->HeadCfg.OSC.PROC_Indx = PROC_OSC;
			m->pCfg->HeadCfg.OSC.VECT_A_Indx = VECT_OSC;
			m->pCfg->HeadCfg.OSC.VECT_B_Indx = VECT_OSC;
			m->pCfg->HeadCfg.OSC.TML_A_Indx = TML_AX_OSC;
			m->pCfg->HeadCfg.OSC.TML_B_Indx = TML_AX_OSC;
			m->pCfg->HeadCfg.OSC.Limits_Harcoded = 0;

			m->pCfg->HeadCfg.OSC.WhelJog_OnlyWhenRun = 0;

			m->pCfg->HeadCfg.OSC.BtnJog_Gain = 4;
			m->pCfg->HeadCfg.OSC.BtnJog_Mode = BTN_JOG_MODE_SINGLE;

			m->pCfg->HeadCfg.OSC.WheelJog_Gain1 = 0.2;
			m->pCfg->HeadCfg.OSC.WhelJog_Mode1 = WHL_JOG_MODE_STEP;

			m->pCfg->HeadCfg.OSC.WheelJog_Gain2 = 0.2;
			m->pCfg->HeadCfg.OSC.WhelJog_Mode2 = WHL_JOG_MODE_STEP;

			m->pCfg->HeadCfg.OSC.DwellDir = 1;

			// WRST
			m->pCfg->HeadCfg.WRST.PROC_Indx = PROC_WRST;
			m->pCfg->HeadCfg.WRST.VECT_A_Indx = VECT_WRST;
			m->pCfg->HeadCfg.WRST.VECT_B_Indx = VECT_WRST;
			m->pCfg->HeadCfg.WRST.TML_A_Indx = TML_AX_WRST;
			m->pCfg->HeadCfg.WRST.TML_B_Indx = TML_AX_WRST;
			m->pCfg->HeadCfg.WRST.Limits_Harcoded = 0;

			m->pCfg->HeadCfg.WRST.BtnJog_Gain = 24.0;
			m->pCfg->HeadCfg.WRST.BtnJog_Mode = BTN_JOG_MODE_SINGLE;

			// AVC
			m->pCfg->HeadCfg.AVC.PROC_Indx = PROC_AVC;
			m->pCfg->HeadCfg.AVC.VECT_A_Indx = VECT_AVC;
			m->pCfg->HeadCfg.AVC.VECT_B_Indx = VECT_AVC;
			m->pCfg->HeadCfg.AVC.TML_A_Indx = TML_AX_AVC;
			m->pCfg->HeadCfg.AVC.TML_B_Indx = TML_AX_AVC;

			m->pCfg->HeadCfg.AVC.BtnJog_Gain = 1;
			m->pCfg->HeadCfg.AVC.BtnJog_Mode = BTN_JOG_MODE_SINGLE;

			// GAS
			m->pCfg->HeadCfg.GAS.PROC_Indx = PROC_GAS;

			// COOL
			m->pCfg->HeadCfg.COOL.PROC_Indx = PROC_COOL;

			// TIG
			m->pCfg->HeadCfg.TIG.PROC_Indx = PROC_TIG_PS;

			// HW
			m->pCfg->HeadCfg.HW.PROC_Indx = PROC_HW_PS;

			// INDX
			m->pCfg->HeadCfg.INDX.PROC_Indx = PROC_INDX;
			m->pCfg->HeadCfg.INDX.VECT_A_Indx = VECT_INDX_1;
			m->pCfg->HeadCfg.INDX.VECT_B_Indx = VECT_INDX_2;
			m->pCfg->HeadCfg.INDX.DC_A_Indx = DC_INDX_1;
			m->pCfg->HeadCfg.INDX.DC_B_Indx = DC_INDX_2;
			m->pCfg->HeadCfg.INDX.BtnJog_Gain = 1.0;

			// WB
			m->pCfg->HeadCfg.WB[WB_UD].PROC_Indx = PROC_WB_UD;
			m->pCfg->HeadCfg.WB[WB_LR].PROC_Indx = PROC_WB_LR;

			m->pCfg->HeadCfg.WB[WB_UD].VECT_Indx = VECT_WB_UD;
			m->pCfg->HeadCfg.WB[WB_LR].VECT_Indx = VECT_WB_LR;

			// Lamp On Off
			m->pCfg->HeadCfg.LampOnOFF.VECT_A_Indx = VECT_OSC + 1;
			m->pCfg->HeadCfg.LampOnOFF.VECT_B_Indx = VECT_WF + 1;

			/////////////////////////////////////////////////////

			// frame size if zero always speed factor is 1.0
			//m->FrameDia = 4.5 * in_2_mm ;
			m->FrameDia = 0.0;

			Configure_SUPER_MINI(m , SUPER_MINI);
			DefaultCalibr_SUPER_MINI(m->pDefaultCalib);

		break;

		/************ BPV_FACE_OSC - 9  ************/
		case BPV_FACE_OSC:

			m->pCfg->HeadCfg.GEN.Torch_Mode = MODE_SINGLE_TORCH;

			// TVL
			m->pCfg->HeadCfg.SwitchHead.VECT_Indx = 0;
			m->pCfg->HeadCfg.SwitchHead.TML_Indx = 0;

			m->pCfg->HeadCfg.TVL.PROC_Indx = PROC_TVL;
			m->pCfg->HeadCfg.TVL.TML_Indx = TML_AX_TVL;

			m->pCfg->HeadCfg.TVL.VECT_Indx = VECT_TVL;
			m->pCfg->HeadCfg.TVL.Enc_Dir = 1;
			//m->pCfg->HeadCfg.TVL.EncPerTick  = 5085;  //  5084.8094458543457034129135792358	// For 1/32 "
			m->pCfg->HeadCfg.TVL.EncPerTick  = 5088; // aby bylo 32 razy
			m->pCfg->HeadCfg.TVL.EncPerTick_SecEnc = 159; // (4000 * 4) / (1" * Pi * 32)
			m->pCfg->HeadCfg.TVL.PinsPerRot = 0;  // Dynamic Configuration
			m->pCfg->HeadCfg.TVL.DistPerTick = 25.4 /32.0; // 1/32"

			m->pCfg->HeadCfg.TVL.BtnJog_Gain = 24;
			m->pCfg->HeadCfg.TVL.BtnJog_Mode = BTN_JOG_MODE_SINGLE;

			// WF
			m->pCfg->HeadCfg.WF.PROC_Indx = PROC_WIRE_FEED;
			m->pCfg->HeadCfg.WF.VECT_A_Indx = VECT_WF;
			m->pCfg->HeadCfg.WF.VECT_B_Indx = VECT_WF_1;
			m->pCfg->HeadCfg.WF.TML_A_Indx = TML_AX_WF;
			m->pCfg->HeadCfg.WF.TML_B_Indx = TML_AX_WF_1;

			m->pCfg->HeadCfg.WF.BtnJog_Gain = 24;
			m->pCfg->HeadCfg.WF.BtnJog_Mode = BTN_JOG_MODE_SINGLE;

			// WP
			m->pCfg->HeadCfg.WP.PROC_Indx = PROC_WIRE_PULSE;
			m->pCfg->HeadCfg.WP.VECT_A_Indx = VECT_WP;
			m->pCfg->HeadCfg.WP.VECT_B_Indx = VECT_WP_1;
			m->pCfg->HeadCfg.WP.TML_A_Indx = TML_AX_WP;
			m->pCfg->HeadCfg.WP.TML_B_Indx = TML_AX_WP_1;

			// OSC
			m->pCfg->HeadCfg.OSC.PROC_Indx = PROC_OSC;
			m->pCfg->HeadCfg.OSC.VECT_A_Indx = VECT_OSC;
			m->pCfg->HeadCfg.OSC.VECT_B_Indx = VECT_OSC;
			m->pCfg->HeadCfg.OSC.TML_A_Indx = TML_AX_OSC;
			m->pCfg->HeadCfg.OSC.TML_B_Indx = TML_AX_OSC;
			m->pCfg->HeadCfg.OSC.Limits_Harcoded = 0;

			m->pCfg->HeadCfg.OSC.WhelJog_OnlyWhenRun = 0;

			m->pCfg->HeadCfg.OSC.BtnJog_Gain = 12;
			m->pCfg->HeadCfg.OSC.BtnJog_Mode = BTN_JOG_MODE_SINGLE;

			m->pCfg->HeadCfg.OSC.WheelJog_Gain1 = 0.2;
			m->pCfg->HeadCfg.OSC.WhelJog_Mode1 = WHL_JOG_MODE_STEP;

			m->pCfg->HeadCfg.OSC.WheelJog_Gain2 = 0.2;
			m->pCfg->HeadCfg.OSC.WhelJog_Mode2 = WHL_JOG_MODE_STEP;

			m->pCfg->HeadCfg.OSC.DwellDir = 1;

			// WRST
			m->pCfg->HeadCfg.WRST.PROC_Indx = PROC_WRST;
			m->pCfg->HeadCfg.WRST.VECT_A_Indx = VECT_WRST;
			m->pCfg->HeadCfg.WRST.VECT_B_Indx = VECT_WRST;
			m->pCfg->HeadCfg.WRST.TML_A_Indx = TML_AX_WRST;
			m->pCfg->HeadCfg.WRST.TML_B_Indx = TML_AX_WRST;
			m->pCfg->HeadCfg.WRST.Limits_Harcoded = 0;

			m->pCfg->HeadCfg.WRST.BtnJog_Gain = 24.0;
			m->pCfg->HeadCfg.WRST.BtnJog_Mode = BTN_JOG_MODE_SINGLE;

			// AVC
			m->pCfg->HeadCfg.AVC.PROC_Indx = PROC_AVC;
			m->pCfg->HeadCfg.AVC.VECT_A_Indx = VECT_AVC;
			m->pCfg->HeadCfg.AVC.VECT_B_Indx = VECT_AVC;
			m->pCfg->HeadCfg.AVC.TML_A_Indx = TML_AX_AVC;
			m->pCfg->HeadCfg.AVC.TML_B_Indx = TML_AX_AVC;

			m->pCfg->HeadCfg.AVC.BtnJog_Gain = 1;
			m->pCfg->HeadCfg.AVC.BtnJog_Mode = BTN_JOG_MODE_SINGLE;

			// GAS
			m->pCfg->HeadCfg.GAS.PROC_Indx = PROC_GAS;

			// COOL
			m->pCfg->HeadCfg.COOL.PROC_Indx = PROC_COOL;

			// TIG
			m->pCfg->HeadCfg.TIG.PROC_Indx = PROC_TIG_PS;

			// HW
			m->pCfg->HeadCfg.HW.PROC_Indx = PROC_HW_PS;

			// INDX
			m->pCfg->HeadCfg.INDX.PROC_Indx = PROC_INDX;
			m->pCfg->HeadCfg.INDX.VECT_A_Indx = VECT_INDX_1;
			m->pCfg->HeadCfg.INDX.VECT_B_Indx = VECT_INDX_2;
			m->pCfg->HeadCfg.INDX.DC_A_Indx = DC_INDX_1;
			m->pCfg->HeadCfg.INDX.DC_B_Indx = DC_INDX_2;
			m->pCfg->HeadCfg.INDX.BtnJog_Gain = 1.0;

			// WB
			m->pCfg->HeadCfg.WB[WB_UD].PROC_Indx = PROC_WB_UD;
			m->pCfg->HeadCfg.WB[WB_LR].PROC_Indx = PROC_WB_LR;

			m->pCfg->HeadCfg.WB[WB_UD].VECT_Indx = VECT_WB_UD;
			m->pCfg->HeadCfg.WB[WB_LR].VECT_Indx = VECT_WB_LR;

			// Lamp On Off
			m->pCfg->HeadCfg.LampOnOFF.VECT_A_Indx = 0; // 0 - not used
			m->pCfg->HeadCfg.LampOnOFF.VECT_B_Indx = 0; // 0 - not used

			/////////////////////////////////////////////////////

			// frame size if zero always speed factor is 1.0
			//m->FrameDia = 4.5 * in_2_mm ;
			m->FrameDia = 0.0;

			Configure_BPV_FACE_OSC(m , BPV_FACE_OSC);
			DefaultCalibr_BPV_FACE_OSC(m->pDefaultCalib);

		break;

		/************ 10 ************/
		case U_BEND_HP_ENC_BEMF:

			m->pCfg->HeadCfg.GEN.Torch_Mode = MODE_SINGLE_TORCH;

			// TVL
			m->pCfg->HeadCfg.SwitchHead.VECT_Indx = 0;
			m->pCfg->HeadCfg.SwitchHead.TML_Indx = 0;

			m->pCfg->HeadCfg.TVL.PROC_Indx = PROC_TVL;
			m->pCfg->HeadCfg.TVL.TML_Indx = TML_AX_TVL;
			m->pCfg->HeadCfg.TVL.DC_Indx = 0;

			m->pCfg->HeadCfg.TVL.VECT_Indx = VECT_TVL;
			m->pCfg->HeadCfg.TVL.Enc_Dir = 1;
			m->pCfg->HeadCfg.TVL.EncPerTick = 200; // (4000 * 4) / (10 * 1/4") * 32 ( becaue 1/32" is one tick")
			m->pCfg->HeadCfg.TVL.PinsPerRot = 640;	// 80 pins , 1/4" per pin
			m->pCfg->HeadCfg.TVL.DistPerTick = 25.4 /32.0; // 1/32"

			m->pCfg->HeadCfg.TVL.BtnJog_Gain = 24;
			m->pCfg->HeadCfg.TVL.BtnJog_Mode = BTN_JOG_MODE_SINGLE;

			// WF
			m->pCfg->HeadCfg.WF.PROC_Indx = PROC_WIRE_FEED;
			m->pCfg->HeadCfg.WF.VECT_A_Indx = VECT_WF;
			m->pCfg->HeadCfg.WF.VECT_B_Indx = VECT_WF_1;
			m->pCfg->HeadCfg.WF.DC_A_Indx = DC_AX_WF;
			m->pCfg->HeadCfg.WF.DC_B_Indx = DC_AX_WF_1;

			m->pCfg->HeadCfg.WF.BtnJog_Gain = 24;
			m->pCfg->HeadCfg.WF.BtnJog_Mode = BTN_JOG_MODE_SINGLE;

			// WP
			m->pCfg->HeadCfg.WP.PROC_Indx = PROC_WIRE_PULSE;
			m->pCfg->HeadCfg.WP.VECT_A_Indx = VECT_WP;
			m->pCfg->HeadCfg.WP.VECT_B_Indx = VECT_WP_1;
			m->pCfg->HeadCfg.WP.DC_A_Indx = DC_AX_WP;
			m->pCfg->HeadCfg.WP.DC_B_Indx = DC_AX_WP_1;

			// OSC
			m->pCfg->HeadCfg.OSC.PROC_Indx = PROC_OSC;
			m->pCfg->HeadCfg.OSC.VECT_A_Indx = VECT_OSC;
			m->pCfg->HeadCfg.OSC.VECT_B_Indx = VECT_OSC;
			m->pCfg->HeadCfg.OSC.TML_A_Indx = TML_AX_OSC;
			m->pCfg->HeadCfg.OSC.TML_B_Indx = TML_AX_OSC;
			m->pCfg->HeadCfg.OSC.Limits_Harcoded = 0;

			m->pCfg->HeadCfg.OSC.BtnJog_Gain = 24.0;
			m->pCfg->HeadCfg.OSC.BtnJog_Mode = BTN_JOG_MODE_SINGLE;

			m->pCfg->HeadCfg.OSC.WheelJog_Gain1 = 5;
			m->pCfg->HeadCfg.OSC.WhelJog_Mode1 = WHL_JOG_MODE_STEP;

			m->pCfg->HeadCfg.OSC.WheelJog_Gain2 = 0.2;
			m->pCfg->HeadCfg.OSC.WhelJog_Mode2 = WHL_JOG_MODE_STEP;
			m->pCfg->HeadCfg.OSC.WhelJog_OnlyWhenRun = 1;

			m->pCfg->HeadCfg.OSC.DwellDir = 1;

			// AVC
			m->pCfg->HeadCfg.AVC.PROC_Indx = PROC_AVC;
			m->pCfg->HeadCfg.AVC.VECT_A_Indx = VECT_AVC;
			m->pCfg->HeadCfg.AVC.VECT_B_Indx = VECT_AVC;
			m->pCfg->HeadCfg.AVC.TML_A_Indx = TML_AX_AVC;
			m->pCfg->HeadCfg.AVC.TML_B_Indx = TML_AX_AVC;

			m->pCfg->HeadCfg.AVC.BtnJog_Gain = 24;
			m->pCfg->HeadCfg.AVC.BtnJog_Mode = BTN_JOG_MODE_SINGLE;

			// GAS
			m->pCfg->HeadCfg.GAS.PROC_Indx = PROC_GAS;

			// COOL
			m->pCfg->HeadCfg.COOL.PROC_Indx = PROC_COOL;

			// TIG
			m->pCfg->HeadCfg.TIG.PROC_Indx = PROC_TIG_PS;

			// HW
			m->pCfg->HeadCfg.HW.PROC_Indx = PROC_HW_PS;

			// INDX
			m->pCfg->HeadCfg.INDX.PROC_Indx = PROC_INDX; // Must be even is disabled

			// WB
			m->pCfg->HeadCfg.WB[WB_UD].PROC_Indx = PROC_WB_UD;
			m->pCfg->HeadCfg.WB[WB_LR].PROC_Indx = PROC_WB_LR;

			m->pCfg->HeadCfg.WB[WB_UD].VECT_Indx = VECT_WB_UD;
			m->pCfg->HeadCfg.WB[WB_LR].VECT_Indx = VECT_WB_LR;

			// Lamp On Off
			m->pCfg->HeadCfg.LampOnOFF.VECT_A_Indx = 0; // 0 - not used
			m->pCfg->HeadCfg.LampOnOFF.VECT_B_Indx = 0; // 0 - not used

			// frame size if zero always speed factor is 1.0
			m->FrameDia = 4.5 * in_2_mm ;
			m->FrameDia = 0.0;

			Configure_U_BEND_HP_ENC_BEMF(m , U_BEND_HP_ENC_BEMF);
			DefaultCalibr_U_BEND_HP_ENC_BEMF(m->pDefaultCalib);

		break;

		/************ 11 ************/
		case F_HEAD_HP_ENC_BEMF:

			m->pCfg->HeadCfg.GEN.Torch_Mode = MODE_SINGLE_TORCH;

			// TVL
			m->pCfg->HeadCfg.SwitchHead.VECT_Indx = 0;
			m->pCfg->HeadCfg.SwitchHead.TML_Indx = 0;

			m->pCfg->HeadCfg.TVL.PROC_Indx = PROC_TVL;
			m->pCfg->HeadCfg.TVL.TML_Indx = TML_AX_TVL;
			m->pCfg->HeadCfg.TVL.DC_Indx = 0;

			m->pCfg->HeadCfg.TVL.VECT_Indx = VECT_TVL;
			m->pCfg->HeadCfg.TVL.Enc_Dir = 1;
			m->pCfg->HeadCfg.TVL.EncPerTick = 38;  // 1/16 inch
			m->pCfg->HeadCfg.TVL.EncPerTick_SecEnc = 38;
			m->pCfg->HeadCfg.TVL.PinsPerRot = 0;  // Dynamic Configuration
			m->pCfg->HeadCfg.TVL.DistPerTick = 25.4 /16.0; // 1/16"

			m->pCfg->HeadCfg.TVL.BtnJog_Gain = 24;
			m->pCfg->HeadCfg.TVL.BtnJog_Mode = BTN_JOG_MODE_SINGLE;

			// WF
			m->pCfg->HeadCfg.WF.PROC_Indx = PROC_WIRE_FEED;
			m->pCfg->HeadCfg.WF.VECT_A_Indx = VECT_WF;
			m->pCfg->HeadCfg.WF.VECT_B_Indx = VECT_WF_1;
			m->pCfg->HeadCfg.WF.DC_A_Indx = DC_AX_WF;
			m->pCfg->HeadCfg.WF.DC_B_Indx = DC_AX_WF_1;

			m->pCfg->HeadCfg.WF.BtnJog_Gain = 24;
			m->pCfg->HeadCfg.WF.BtnJog_Mode = BTN_JOG_MODE_SINGLE;

			// WP
			m->pCfg->HeadCfg.WP.PROC_Indx = PROC_WIRE_PULSE;
			m->pCfg->HeadCfg.WP.VECT_A_Indx = VECT_WP;
			m->pCfg->HeadCfg.WP.VECT_B_Indx = VECT_WP_1;
			m->pCfg->HeadCfg.WP.DC_A_Indx = DC_AX_WP;
			m->pCfg->HeadCfg.WP.DC_B_Indx = DC_AX_WP_1;

			// OSC
			m->pCfg->HeadCfg.OSC.PROC_Indx = PROC_OSC;
			m->pCfg->HeadCfg.OSC.VECT_A_Indx = VECT_OSC;
			m->pCfg->HeadCfg.OSC.VECT_B_Indx = VECT_OSC;
			m->pCfg->HeadCfg.OSC.TML_A_Indx = TML_AX_OSC;
			m->pCfg->HeadCfg.OSC.TML_B_Indx = TML_AX_OSC;
			m->pCfg->HeadCfg.OSC.Limits_Harcoded = 0;

			m->pCfg->HeadCfg.OSC.BtnJog_Gain = 24.0;
			m->pCfg->HeadCfg.OSC.BtnJog_Mode = BTN_JOG_MODE_SINGLE;

			m->pCfg->HeadCfg.OSC.WheelJog_Gain1 = 5.0;
			m->pCfg->HeadCfg.OSC.WhelJog_Mode1 = WHL_JOG_MODE_STEP;

			m->pCfg->HeadCfg.OSC.WheelJog_Gain2 = 0.2;
			m->pCfg->HeadCfg.OSC.WhelJog_Mode2 = WHL_JOG_MODE_STEP;
			m->pCfg->HeadCfg.OSC.WhelJog_OnlyWhenRun = 1;

			m->pCfg->HeadCfg.OSC.DwellDir = 1;

			// AVC
			m->pCfg->HeadCfg.AVC.PROC_Indx = PROC_AVC;
			m->pCfg->HeadCfg.AVC.VECT_A_Indx = VECT_AVC;
			m->pCfg->HeadCfg.AVC.VECT_B_Indx = VECT_AVC;
			m->pCfg->HeadCfg.AVC.TML_A_Indx = TML_AX_AVC;
			m->pCfg->HeadCfg.AVC.TML_B_Indx = TML_AX_AVC;

			m->pCfg->HeadCfg.AVC.BtnJog_Gain = 24;
			m->pCfg->HeadCfg.AVC.BtnJog_Mode = BTN_JOG_MODE_SINGLE;

			// GAS
			m->pCfg->HeadCfg.GAS.PROC_Indx = PROC_GAS;

			// COOL
			m->pCfg->HeadCfg.COOL.PROC_Indx = PROC_COOL;

			// TIG
			m->pCfg->HeadCfg.TIG.PROC_Indx = PROC_TIG_PS;

			// HW
			m->pCfg->HeadCfg.HW.PROC_Indx = PROC_HW_PS;

			// INDX
			m->pCfg->HeadCfg.INDX.PROC_Indx = PROC_INDX; // Must be even is disabled

			// WB
			m->pCfg->HeadCfg.WB[WB_UD].PROC_Indx = PROC_WB_UD;
			m->pCfg->HeadCfg.WB[WB_LR].PROC_Indx = PROC_WB_LR;

			m->pCfg->HeadCfg.WB[WB_UD].VECT_Indx = VECT_WB_UD;
			m->pCfg->HeadCfg.WB[WB_LR].VECT_Indx = VECT_WB_LR;

			// Lamp On Off
			m->pCfg->HeadCfg.LampOnOFF.VECT_A_Indx = 0; // 0 - not used
			m->pCfg->HeadCfg.LampOnOFF.VECT_B_Indx = 0; // 0 - not used

			/////////////////////////////////////////////////////

			// frame size if zero always speed factor is 1.0
			//m->FrameDia = 4.5 * in_2_mm ;
			m->FrameDia = 0.0;

			Configure_F_HEAD_HP_ENC_BEMF(m , F_HEAD_HP_ENCODER);
			DefaultCalibr_F_HEAD_HP_ENC_BEMF(m->pDefaultCalib);

		break;

		/************ BPV_FACE_OSC_ENC - 12  ************/
		case BPV_FACE_OSC_ENC:

			m->pCfg->HeadCfg.GEN.Torch_Mode = MODE_SINGLE_TORCH;

			// TVL
			m->pCfg->HeadCfg.SwitchHead.VECT_Indx = 0;
			m->pCfg->HeadCfg.SwitchHead.TML_Indx = 0;

			m->pCfg->HeadCfg.TVL.PROC_Indx = PROC_TVL;
			m->pCfg->HeadCfg.TVL.TML_Indx = TML_AX_TVL;

			m->pCfg->HeadCfg.TVL.VECT_Indx = VECT_TVL;
			m->pCfg->HeadCfg.TVL.Enc_Dir = 1;
			//m->pCfg->HeadCfg.TVL.EncPerTick  = 5085;  //  5084.8094458543457034129135792358	// For 1/32 "
			m->pCfg->HeadCfg.TVL.EncPerTick  = 5088; // aby bylo 32 razy
			m->pCfg->HeadCfg.TVL.EncPerTick_SecEnc = 159; // (4000 * 4) / (1" * Pi * 32)
			m->pCfg->HeadCfg.TVL.PinsPerRot = 0;  // Dynamic Configuration
			m->pCfg->HeadCfg.TVL.DistPerTick = 25.4 /32.0; // 1/32"

			m->pCfg->HeadCfg.TVL.BtnJog_Gain = 24;
			m->pCfg->HeadCfg.TVL.BtnJog_Mode = BTN_JOG_MODE_SINGLE;

			// WF
			m->pCfg->HeadCfg.WF.PROC_Indx = PROC_WIRE_FEED;
			m->pCfg->HeadCfg.WF.VECT_A_Indx = VECT_WF;
			m->pCfg->HeadCfg.WF.VECT_B_Indx = VECT_WF_1;
			m->pCfg->HeadCfg.WF.TML_A_Indx = TML_AX_WF;
			m->pCfg->HeadCfg.WF.TML_B_Indx = TML_AX_WF_1;

			m->pCfg->HeadCfg.WF.BtnJog_Gain = 24;
			m->pCfg->HeadCfg.WF.BtnJog_Mode = BTN_JOG_MODE_SINGLE;

			// WP
			m->pCfg->HeadCfg.WP.PROC_Indx = PROC_WIRE_PULSE;
			m->pCfg->HeadCfg.WP.VECT_A_Indx = VECT_WP;
			m->pCfg->HeadCfg.WP.VECT_B_Indx = VECT_WP_1;
			m->pCfg->HeadCfg.WP.TML_A_Indx = TML_AX_WP;
			m->pCfg->HeadCfg.WP.TML_B_Indx = TML_AX_WP_1;

			// OSC
			m->pCfg->HeadCfg.OSC.PROC_Indx = PROC_OSC;
			m->pCfg->HeadCfg.OSC.VECT_A_Indx = VECT_OSC;
			m->pCfg->HeadCfg.OSC.VECT_B_Indx = VECT_OSC;
			m->pCfg->HeadCfg.OSC.TML_A_Indx = TML_AX_OSC;
			m->pCfg->HeadCfg.OSC.TML_B_Indx = TML_AX_OSC;
			m->pCfg->HeadCfg.OSC.Limits_Harcoded = 0;

			m->pCfg->HeadCfg.OSC.WhelJog_OnlyWhenRun = 0;

			m->pCfg->HeadCfg.OSC.BtnJog_Gain = 12;
			m->pCfg->HeadCfg.OSC.BtnJog_Mode = BTN_JOG_MODE_SINGLE;

			m->pCfg->HeadCfg.OSC.WheelJog_Gain1 = 0.2;
			m->pCfg->HeadCfg.OSC.WhelJog_Mode1 = WHL_JOG_MODE_STEP;

			m->pCfg->HeadCfg.OSC.WheelJog_Gain2 = 0.2;
			m->pCfg->HeadCfg.OSC.WhelJog_Mode2 = WHL_JOG_MODE_STEP;

			m->pCfg->HeadCfg.OSC.DwellDir = 1;

			// WRST
			m->pCfg->HeadCfg.WRST.PROC_Indx = PROC_WRST;
			m->pCfg->HeadCfg.WRST.VECT_A_Indx = VECT_WRST;
			m->pCfg->HeadCfg.WRST.VECT_B_Indx = VECT_WRST;
			m->pCfg->HeadCfg.WRST.TML_A_Indx = TML_AX_WRST;
			m->pCfg->HeadCfg.WRST.TML_B_Indx = TML_AX_WRST;
			m->pCfg->HeadCfg.WRST.Limits_Harcoded = 0;

			m->pCfg->HeadCfg.WRST.BtnJog_Gain = 24.0;
			m->pCfg->HeadCfg.WRST.BtnJog_Mode = BTN_JOG_MODE_SINGLE;

			// AVC
			m->pCfg->HeadCfg.AVC.PROC_Indx = PROC_AVC;
			m->pCfg->HeadCfg.AVC.VECT_A_Indx = VECT_AVC;
			m->pCfg->HeadCfg.AVC.VECT_B_Indx = VECT_AVC;
			m->pCfg->HeadCfg.AVC.TML_A_Indx = TML_AX_AVC;
			m->pCfg->HeadCfg.AVC.TML_B_Indx = TML_AX_AVC;

			m->pCfg->HeadCfg.AVC.BtnJog_Gain = 1;
			m->pCfg->HeadCfg.AVC.BtnJog_Mode = BTN_JOG_MODE_SINGLE;

			// GAS
			m->pCfg->HeadCfg.GAS.PROC_Indx = PROC_GAS;

			// COOL
			m->pCfg->HeadCfg.COOL.PROC_Indx = PROC_COOL;

			// TIG
			m->pCfg->HeadCfg.TIG.PROC_Indx = PROC_TIG_PS;

			// HW
			m->pCfg->HeadCfg.HW.PROC_Indx = PROC_HW_PS;

			// INDX
			m->pCfg->HeadCfg.INDX.PROC_Indx = PROC_INDX;
			m->pCfg->HeadCfg.INDX.VECT_A_Indx = VECT_INDX_1;
			m->pCfg->HeadCfg.INDX.VECT_B_Indx = VECT_INDX_2;
			m->pCfg->HeadCfg.INDX.DC_A_Indx = DC_INDX_1;
			m->pCfg->HeadCfg.INDX.DC_B_Indx = DC_INDX_2;
			m->pCfg->HeadCfg.INDX.BtnJog_Gain = 1.0;

			// WB
			m->pCfg->HeadCfg.WB[WB_UD].PROC_Indx = PROC_WB_UD;
			m->pCfg->HeadCfg.WB[WB_LR].PROC_Indx = PROC_WB_LR;

			m->pCfg->HeadCfg.WB[WB_UD].VECT_Indx = VECT_WB_UD;
			m->pCfg->HeadCfg.WB[WB_LR].VECT_Indx = VECT_WB_LR;

			// Lamp On Off
			m->pCfg->HeadCfg.LampOnOFF.VECT_A_Indx = 0; // 0 - not used
			m->pCfg->HeadCfg.LampOnOFF.VECT_B_Indx = 0; // 0 - not used

			/////////////////////////////////////////////////////

			// frame size if zero always speed factor is 1.0
			//m->FrameDia = 4.5 * in_2_mm ;
			m->FrameDia = 0.0;

			Configure_BPV_FACE_OSC_ENC(m , BPV_FACE_OSC_ENC);
			DefaultCalibr_BPV_FACE_OSC(m->pDefaultCalib);

		break;

		/************ BPV_FACE_OSC_EXP - 13  ************/
		case BPV_FACE_OSC_EXP:
		/************ BPV2_FACE_OSC_EXP - 27  ************/
		case BPV2_FACE_OSC_EXP:

			m->pCfg->HeadCfg.GEN.Torch_Mode = MODE_SINGLE_TORCH;

			// TVL
			m->pCfg->HeadCfg.SwitchHead.VECT_Indx = 0;
			m->pCfg->HeadCfg.SwitchHead.TML_Indx = 0;

			m->pCfg->HeadCfg.TVL.PROC_Indx = PROC_TVL;
			m->pCfg->HeadCfg.TVL.TML_Indx = TML_AX_TVL;

			m->pCfg->HeadCfg.TVL.VECT_Indx = VECT_TVL;
			m->pCfg->HeadCfg.TVL.Enc_Dir = 1;
			//m->pCfg->HeadCfg.TVL.EncPerTick  = 5085;  //  5084.8094458543457034129135792358	// For 1/32 "
			m->pCfg->HeadCfg.TVL.EncPerTick  = 5088; // aby bylo 32 razy
			m->pCfg->HeadCfg.TVL.EncPerTick_SecEnc = 159; // (4000 * 4) / (1" * Pi * 32)
			m->pCfg->HeadCfg.TVL.PinsPerRot = 0;  // Dynamic Configuration
			m->pCfg->HeadCfg.TVL.DistPerTick = 25.4 /32.0; // 1/32"

			m->pCfg->HeadCfg.TVL.BtnJog_Gain = 24;
			m->pCfg->HeadCfg.TVL.BtnJog_Mode = BTN_JOG_MODE_SINGLE;

			// WF
			m->pCfg->HeadCfg.WF.PROC_Indx = PROC_WIRE_FEED;
			m->pCfg->HeadCfg.WF.VECT_A_Indx = VECT_WF;
			m->pCfg->HeadCfg.WF.VECT_B_Indx = VECT_WF_1;
			m->pCfg->HeadCfg.WF.TML_A_Indx = TML_AX_WF;
			m->pCfg->HeadCfg.WF.TML_B_Indx = TML_AX_WF_1;

			m->pCfg->HeadCfg.WF.BtnJog_Gain = 24;
			m->pCfg->HeadCfg.WF.BtnJog_Mode = BTN_JOG_MODE_SINGLE;

			// WP
			m->pCfg->HeadCfg.WP.PROC_Indx = PROC_WIRE_PULSE;
			m->pCfg->HeadCfg.WP.VECT_A_Indx = VECT_WP;
			m->pCfg->HeadCfg.WP.VECT_B_Indx = VECT_WP_1;
			m->pCfg->HeadCfg.WP.TML_A_Indx = TML_AX_WP;
			m->pCfg->HeadCfg.WP.TML_B_Indx = TML_AX_WP_1;

			// OSC
			m->pCfg->HeadCfg.OSC.PROC_Indx = PROC_OSC;
			m->pCfg->HeadCfg.OSC.VECT_A_Indx = VECT_OSC;
			m->pCfg->HeadCfg.OSC.VECT_B_Indx = VECT_OSC;
			m->pCfg->HeadCfg.OSC.TML_A_Indx = TML_AX_OSC;
			m->pCfg->HeadCfg.OSC.TML_B_Indx = TML_AX_OSC;
			m->pCfg->HeadCfg.OSC.Limits_Harcoded = 0;

			m->pCfg->HeadCfg.OSC.WhelJog_OnlyWhenRun = 0;

			m->pCfg->HeadCfg.OSC.BtnJog_Gain = 12;
			m->pCfg->HeadCfg.OSC.BtnJog_Mode = BTN_JOG_MODE_SINGLE;

			m->pCfg->HeadCfg.OSC.WheelJog_Gain1 = 0.2;
			m->pCfg->HeadCfg.OSC.WhelJog_Mode1 = WHL_JOG_MODE_STEP;

			m->pCfg->HeadCfg.OSC.WheelJog_Gain2 = 0.2;
			m->pCfg->HeadCfg.OSC.WhelJog_Mode2 = WHL_JOG_MODE_STEP;

			m->pCfg->HeadCfg.OSC.DwellDir = 1;

			// WRST
			m->pCfg->HeadCfg.WRST.PROC_Indx = PROC_WRST;
			m->pCfg->HeadCfg.WRST.VECT_A_Indx = VECT_WRST;
			m->pCfg->HeadCfg.WRST.VECT_B_Indx = VECT_WRST;
			m->pCfg->HeadCfg.WRST.TML_A_Indx = TML_AX_WRST;
			m->pCfg->HeadCfg.WRST.TML_B_Indx = TML_AX_WRST;
			m->pCfg->HeadCfg.WRST.Limits_Harcoded = 0;

			m->pCfg->HeadCfg.WRST.BtnJog_Gain = 24.0;
			m->pCfg->HeadCfg.WRST.BtnJog_Mode = BTN_JOG_MODE_SINGLE;

			// AVC
			m->pCfg->HeadCfg.AVC.PROC_Indx = PROC_AVC;
			m->pCfg->HeadCfg.AVC.VECT_A_Indx = VECT_AVC;
			m->pCfg->HeadCfg.AVC.VECT_B_Indx = VECT_AVC;
			m->pCfg->HeadCfg.AVC.TML_A_Indx = TML_AX_AVC;
			m->pCfg->HeadCfg.AVC.TML_B_Indx = TML_AX_AVC;

			m->pCfg->HeadCfg.AVC.BtnJog_Gain = 1;
			m->pCfg->HeadCfg.AVC.BtnJog_Mode = BTN_JOG_MODE_SINGLE;

			// GAS
			m->pCfg->HeadCfg.GAS.PROC_Indx = PROC_GAS;

			// COOL
			m->pCfg->HeadCfg.COOL.PROC_Indx = PROC_COOL;

			// TIG
			m->pCfg->HeadCfg.TIG.PROC_Indx = PROC_TIG_PS;

			// HW
			m->pCfg->HeadCfg.HW.PROC_Indx = PROC_HW_PS;

			// INDX
			m->pCfg->HeadCfg.INDX.PROC_Indx = PROC_INDX;
			m->pCfg->HeadCfg.INDX.VECT_A_Indx = VECT_INDX_1;
			m->pCfg->HeadCfg.INDX.VECT_B_Indx = VECT_INDX_2;
			m->pCfg->HeadCfg.INDX.DC_A_Indx = DC_INDX_1;
			m->pCfg->HeadCfg.INDX.DC_B_Indx = DC_INDX_2;
			m->pCfg->HeadCfg.INDX.BtnJog_Gain = 1.0;

			// WB
			m->pCfg->HeadCfg.WB[WB_UD].PROC_Indx = PROC_WB_UD;
			m->pCfg->HeadCfg.WB[WB_LR].PROC_Indx = PROC_WB_LR;

			m->pCfg->HeadCfg.WB[WB_UD].VECT_Indx = VECT_WB_UD;
			m->pCfg->HeadCfg.WB[WB_LR].VECT_Indx = VECT_WB_LR;

			// Lamp On Off
			m->pCfg->HeadCfg.LampOnOFF.VECT_A_Indx = 0; // 0 - not used
			m->pCfg->HeadCfg.LampOnOFF.VECT_B_Indx = 0; // 0 - not used

			/////////////////////////////////////////////////////

			// frame size if zero always speed factor is 1.0
			//m->FrameDia = 4.5 * in_2_mm ;
			m->FrameDia = 0.0;

			switch(headType){

				case BPV_FACE_OSC_EXP:
					Configure_BPV_FACE_OSC_EXP(m , BPV_FACE_OSC_EXP);
				break;

				case BPV2_FACE_OSC_EXP:
					Configure_BPV2_FACE_OSC_EXP(m , BPV2_FACE_OSC_EXP);
				break;
			}

			DefaultCalibr_BPV_FACE_OSC(m->pDefaultCalib);

		break;

		/************ 14 ************/
		case M_94:

			m->pCfg->HeadCfg.GEN.Torch_Mode = MODE_SINGLE_TORCH;

			// TVL
			m->pCfg->HeadCfg.SwitchHead.VECT_Indx = 0;
			m->pCfg->HeadCfg.SwitchHead.TML_Indx = 0;

			m->pCfg->HeadCfg.TVL.PROC_Indx = PROC_TVL;
			m->pCfg->HeadCfg.TVL.TML_Indx = TML_AX_TVL;

			m->pCfg->HeadCfg.TVL.VECT_Indx = VECT_TVL;
			m->pCfg->HeadCfg.TVL.Enc_Dir = 1;
			//m->pCfg->HeadCfg.TVL.EncPerTick  = 5085;  //  5084.8094458543457034129135792358	// For 1/32 "
			m->pCfg->HeadCfg.TVL.EncPerTick  = 5088; // aby bylo 32 razy
			m->pCfg->HeadCfg.TVL.EncPerTick_SecEnc = 159; // (4000 * 4) / (1" * Pi * 32)
			m->pCfg->HeadCfg.TVL.PinsPerRot = 0;  // Dynamic Configuration
			m->pCfg->HeadCfg.TVL.DistPerTick = 25.4 /32.0; // 1/32"

			m->pCfg->HeadCfg.TVL.BtnJog_Gain = 24;
			m->pCfg->HeadCfg.TVL.BtnJog_Mode = BTN_JOG_MODE_SINGLE;

			// WF
			m->pCfg->HeadCfg.WF.PROC_Indx = PROC_WIRE_FEED;
			m->pCfg->HeadCfg.WF.VECT_A_Indx = VECT_WF;
			m->pCfg->HeadCfg.WF.VECT_B_Indx = VECT_WF_1;
			m->pCfg->HeadCfg.WF.DC_A_Indx = DC_AX_WF;
			m->pCfg->HeadCfg.WF.DC_B_Indx = DC_AX_WF_1;

			m->pCfg->HeadCfg.WF.BtnJog_Gain = 24;
			m->pCfg->HeadCfg.WF.BtnJog_Mode = BTN_JOG_MODE_SINGLE;

			// WP
			m->pCfg->HeadCfg.WP.PROC_Indx = PROC_WIRE_PULSE;
			m->pCfg->HeadCfg.WP.VECT_A_Indx = VECT_WP;
			m->pCfg->HeadCfg.WP.VECT_B_Indx = VECT_WP_1;
			m->pCfg->HeadCfg.WP.DC_A_Indx = DC_AX_WP;
			m->pCfg->HeadCfg.WP.DC_B_Indx = DC_AX_WP_1;

			// OSC
			m->pCfg->HeadCfg.OSC.PROC_Indx = PROC_OSC;
			m->pCfg->HeadCfg.OSC.VECT_A_Indx = VECT_OSC;
			m->pCfg->HeadCfg.OSC.VECT_B_Indx = VECT_OSC;
			m->pCfg->HeadCfg.OSC.TML_A_Indx = TML_AX_OSC;
			m->pCfg->HeadCfg.OSC.TML_B_Indx = TML_AX_OSC;
			m->pCfg->HeadCfg.OSC.Limits_Harcoded = 0;

			m->pCfg->HeadCfg.OSC.WhelJog_OnlyWhenRun = 0;

			m->pCfg->HeadCfg.OSC.BtnJog_Gain = 4;
			m->pCfg->HeadCfg.OSC.BtnJog_Mode = BTN_JOG_MODE_SINGLE;

			m->pCfg->HeadCfg.OSC.WheelJog_Gain1 = 0.2;
			m->pCfg->HeadCfg.OSC.WhelJog_Mode1 = WHL_JOG_MODE_STEP;

			m->pCfg->HeadCfg.OSC.WheelJog_Gain2 = 0.2;
			m->pCfg->HeadCfg.OSC.WhelJog_Mode2 = WHL_JOG_MODE_STEP;

			m->pCfg->HeadCfg.OSC.DwellDir = 1;

			// WRST
			m->pCfg->HeadCfg.WRST.PROC_Indx = PROC_WRST;
			m->pCfg->HeadCfg.WRST.VECT_A_Indx = VECT_WRST;
			m->pCfg->HeadCfg.WRST.VECT_B_Indx = VECT_WRST;
			m->pCfg->HeadCfg.WRST.TML_A_Indx = TML_AX_WRST;
			m->pCfg->HeadCfg.WRST.TML_B_Indx = TML_AX_WRST;
			m->pCfg->HeadCfg.WRST.Limits_Harcoded = 0;

			m->pCfg->HeadCfg.WRST.BtnJog_Gain = 24.0;
			m->pCfg->HeadCfg.WRST.BtnJog_Mode = BTN_JOG_MODE_SINGLE;

			// AVC
			m->pCfg->HeadCfg.AVC.PROC_Indx = PROC_AVC;
			m->pCfg->HeadCfg.AVC.VECT_A_Indx = VECT_AVC;
			m->pCfg->HeadCfg.AVC.VECT_B_Indx = VECT_AVC;
			m->pCfg->HeadCfg.AVC.TML_A_Indx = TML_AX_AVC;
			m->pCfg->HeadCfg.AVC.TML_B_Indx = TML_AX_AVC;

			m->pCfg->HeadCfg.AVC.BtnJog_Gain = 1;
			m->pCfg->HeadCfg.AVC.BtnJog_Mode = BTN_JOG_MODE_SINGLE;

			// GAS
			m->pCfg->HeadCfg.GAS.PROC_Indx = PROC_GAS;

			// COOL
			m->pCfg->HeadCfg.COOL.PROC_Indx = PROC_COOL;

			// TIG
			m->pCfg->HeadCfg.TIG.PROC_Indx = PROC_TIG_PS;

			// HW
			m->pCfg->HeadCfg.HW.PROC_Indx = PROC_HW_PS;

			// INDX
			m->pCfg->HeadCfg.INDX.PROC_Indx = PROC_INDX;
			m->pCfg->HeadCfg.INDX.VECT_A_Indx = VECT_INDX_1;
			m->pCfg->HeadCfg.INDX.VECT_B_Indx = VECT_INDX_2;
			m->pCfg->HeadCfg.INDX.DC_A_Indx = DC_INDX_1;
			m->pCfg->HeadCfg.INDX.DC_B_Indx = DC_INDX_2;
			m->pCfg->HeadCfg.INDX.BtnJog_Gain = 1.0;

			// WB
			m->pCfg->HeadCfg.WB[WB_UD].PROC_Indx = PROC_WB_UD;
			m->pCfg->HeadCfg.WB[WB_LR].PROC_Indx = PROC_WB_LR;

			m->pCfg->HeadCfg.WB[WB_UD].VECT_Indx = VECT_WB_UD;
			m->pCfg->HeadCfg.WB[WB_LR].VECT_Indx = VECT_WB_LR;

			// Lamp On Off
			m->pCfg->HeadCfg.LampOnOFF.VECT_A_Indx = 0; // 0 - not used
			m->pCfg->HeadCfg.LampOnOFF.VECT_B_Indx = 0; // 0 - not used

			/////////////////////////////////////////////////////

			// frame size if zero always speed factor is 1.0
			//m->FrameDia = 4.5 * in_2_mm ;
			m->FrameDia = 0.0;

			Configure_M_94(m , M_94);
			DefaultCalibr_M_94(m->pDefaultCalib);

		break;

///////////////////////////////////////
///////  BPV Ver 2 Heads
//////////////////////////////////////

		/************ BPV_v2 - 15 ************/
		/************ BPV_v2_TT_BO - 19 ************/
		case BPV_v2:
		case BPV_v2_Video:
		case BPV_v2_TT_BO:
		case MIG_TIG_HEAD:

			m->pCfg->HeadCfg.GEN.Torch_Mode = MODE_SINGLE_TORCH;

			// TVL
			m->pCfg->HeadCfg.SwitchHead.VECT_Indx = VECT_TVL;
			m->pCfg->HeadCfg.SwitchHead.TML_Indx = TML_AX_TVL;

			m->pCfg->HeadCfg.TVL.PROC_Indx = PROC_TVL;
			m->pCfg->HeadCfg.TVL.TML_Indx = TML_AX_TVL;

			// This is like BPV
			m->pCfg->HeadCfg.TVL.VECT_Indx = VECT_TVL;
			m->pCfg->HeadCfg.TVL.Enc_Dir = 1;
			//m->pCfg->HeadCfg.TVL.EncPerTick  = 5085;  //  5084.8094458543457034129135792358	// For 1/32 "
			m->pCfg->HeadCfg.TVL.EncPerTick  = 5088; // aby bylo 32 razy
			m->pCfg->HeadCfg.TVL.EncPerTick_SecEnc = 159; // (4000 * 4) / (1" * Pi * 32)
			m->pCfg->HeadCfg.TVL.PinsPerRot = 0;  // Dynamic Configuration
			m->pCfg->HeadCfg.TVL.DistPerTick = 25.4 /32.0; // 1/32"
			/////////////////////

			m->pCfg->HeadCfg.TVL.BtnJog_Gain = 24;
			m->pCfg->HeadCfg.TVL.BtnJog_Mode = BTN_JOG_MODE_SINGLE;

			// I took it from BPV Head
			// WF
			m->pCfg->HeadCfg.WF.PROC_Indx = PROC_WIRE_FEED;
			m->pCfg->HeadCfg.WF.VECT_A_Indx = VECT_WF;
			m->pCfg->HeadCfg.WF.VECT_B_Indx = VECT_WF_1;
			m->pCfg->HeadCfg.WF.TML_A_Indx = TML_AX_WF;
			m->pCfg->HeadCfg.WF.TML_B_Indx = TML_AX_WF_1;

			m->pCfg->HeadCfg.WF.VECT_Aux_A_Indx = VECT_AUX_WF;
			m->pCfg->HeadCfg.WF.VECT_Aux_B_Indx = VECT_AUX_WF_1;
			m->pCfg->HeadCfg.WF.TML_Aux_A_Indx = TML_AUX_AX_WF;
			m->pCfg->HeadCfg.WF.TML_Aux_B_Indx = TML_AUX_AX_WF_1;

			m->pCfg->HeadCfg.WF.BtnJog_Gain = 24;
			m->pCfg->HeadCfg.WF.BtnJog_Mode = BTN_JOG_MODE_SINGLE;

			// WP
			m->pCfg->HeadCfg.WP.PROC_Indx = PROC_WIRE_PULSE;
			m->pCfg->HeadCfg.WP.VECT_A_Indx = VECT_WP;
			m->pCfg->HeadCfg.WP.VECT_B_Indx = VECT_WP_1;
			m->pCfg->HeadCfg.WP.TML_A_Indx = TML_AX_WP;
			m->pCfg->HeadCfg.WP.TML_B_Indx = TML_AX_WP_1;

			// OSC
			m->pCfg->HeadCfg.OSC.PROC_Indx = PROC_OSC;
			m->pCfg->HeadCfg.OSC.VECT_A_Indx = VECT_OSC;
			m->pCfg->HeadCfg.OSC.VECT_B_Indx = VECT_OSC;
			m->pCfg->HeadCfg.OSC.TML_A_Indx = TML_AX_OSC;
			m->pCfg->HeadCfg.OSC.TML_B_Indx = TML_AX_OSC;
			m->pCfg->HeadCfg.OSC.Limits_Harcoded = 0;

			m->pCfg->HeadCfg.OSC.WhelJog_OnlyWhenRun = 0;

			m->pCfg->HeadCfg.OSC.BtnJog_Gain = 4;
			m->pCfg->HeadCfg.OSC.BtnJog_Mode = BTN_JOG_MODE_SINGLE;

			m->pCfg->HeadCfg.OSC.WheelJog_Gain1 = 0.2;
			m->pCfg->HeadCfg.OSC.WhelJog_Mode1 = WHL_JOG_MODE_STEP;

			m->pCfg->HeadCfg.OSC.WheelJog_Gain2 = 0.2;
			m->pCfg->HeadCfg.OSC.WhelJog_Mode2 = WHL_JOG_MODE_STEP;

			m->pCfg->HeadCfg.OSC.DwellDir = 1;

			// WRST
			m->pCfg->HeadCfg.WRST.PROC_Indx = PROC_WRST;
			m->pCfg->HeadCfg.WRST.VECT_A_Indx = VECT_WRST;
			m->pCfg->HeadCfg.WRST.VECT_B_Indx = VECT_WRST;
			m->pCfg->HeadCfg.WRST.TML_A_Indx = TML_AX_WRST;
			m->pCfg->HeadCfg.WRST.TML_B_Indx = TML_AX_WRST;
			m->pCfg->HeadCfg.WRST.Limits_Harcoded = 0;

			m->pCfg->HeadCfg.WRST.BtnJog_Gain = 24.0;
			m->pCfg->HeadCfg.WRST.BtnJog_Mode = BTN_JOG_MODE_SINGLE;

			// AVC
			m->pCfg->HeadCfg.AVC.PROC_Indx = PROC_AVC;
			m->pCfg->HeadCfg.AVC.VECT_A_Indx = VECT_AVC;
			m->pCfg->HeadCfg.AVC.VECT_B_Indx = VECT_AVC;
			m->pCfg->HeadCfg.AVC.TML_A_Indx = TML_AX_AVC;
			m->pCfg->HeadCfg.AVC.TML_B_Indx = TML_AX_AVC;

			m->pCfg->HeadCfg.AVC.BtnJog_Gain = 1;
			m->pCfg->HeadCfg.AVC.BtnJog_Mode = BTN_JOG_MODE_SINGLE;

			// INDX
			m->pCfg->HeadCfg.INDX.PROC_Indx = PROC_INDX;
			m->pCfg->HeadCfg.INDX.VECT_A_Indx = VECT_INDX_1;
			m->pCfg->HeadCfg.INDX.VECT_B_Indx = VECT_INDX_2;
			m->pCfg->HeadCfg.INDX.TML_A_Indx = TML_AX_INDX;
			m->pCfg->HeadCfg.INDX.TML_B_Indx = TML_AX_INDX_1;
			m->pCfg->HeadCfg.INDX.BtnJog_Gain = 1.0;

			// GAS
			m->pCfg->HeadCfg.GAS.PROC_Indx = PROC_GAS;

			// COOL
			m->pCfg->HeadCfg.COOL.PROC_Indx = PROC_COOL;

			// TIG
			m->pCfg->HeadCfg.TIG.PROC_Indx = PROC_TIG_PS;

			// HW
			m->pCfg->HeadCfg.HW.PROC_Indx = PROC_HW_PS;

			if(headType != MIG_TIG_HEAD){

				// WB
				m->pCfg->HeadCfg.WB[WB_UD].PROC_Indx = PROC_WB_UD;
				m->pCfg->HeadCfg.WB[WB_LR].PROC_Indx = PROC_WB_LR;

				m->pCfg->HeadCfg.WB[WB_UD].VECT_Indx = VECT_WB_UD;
				m->pCfg->HeadCfg.WB[WB_LR].VECT_Indx = VECT_WB_LR;

				// Lamp On Off
				m->pCfg->HeadCfg.LampOnOFF.VECT_A_Indx = VECT_OSC + 1;
				m->pCfg->HeadCfg.LampOnOFF.VECT_B_Indx = VECT_INDX_1 + 1;

			}

			/////////////////////////////////////////////////////

			// frame size if zero always speed factor is 1.0
			//m->FrameDia = 4.5 * in_2_mm ;
			m->FrameDia = 0.0;

			switch(headType){

				case BPV_v2:
				case BPV_v2_Video:

					Configure_BPV_v2(m , headType);
					DefaultCalibr_BPV_v2(m->pDefaultCalib);

				break;

				case BPV_v2_TT_BO:

					Configure_BPV_v2_TT_BO(m , headType);
					DefaultCalibr_BPV_v2_TT_BO(m->pDefaultCalib);

				break;

				case MIG_TIG_HEAD:

					m->pCfg->HeadCfg.OSC.BtnJog_Gain = 20.0;

					m->pCfg->HeadCfg.INDX.VECT_B_Indx = 0;
					m->pCfg->HeadCfg.INDX.TML_B_Indx = 0;

					m->pCfg->HeadCfg.WF.VECT_B_Indx = m->pCfg->HeadCfg.WF.VECT_A_Indx;
					m->pCfg->HeadCfg.WF.TML_B_Indx = m->pCfg->HeadCfg.WF.TML_A_Indx;

					m->pCfg->HeadCfg.WP.VECT_B_Indx = m->pCfg->HeadCfg.WP.VECT_A_Indx;
					m->pCfg->HeadCfg.WP.TML_B_Indx = m->pCfg->HeadCfg.WP.TML_A_Indx;

					Configure_MIG_TIG(m , headType);
					DefaultCalibr_MIG_TIG(m->pDefaultCalib);

				break;

			}

		break;

		/************ BPV_v2_MPBO - 16 ************/
		/************ BPV_v2_MT_BO - 20 ************/
		/************ BPV_v2_MT - 28 ************/
		case BPV_v2_MPBO:
		case BPV_v2_MT_BO:
		case BPV_v2_MT:

			m->pCfg->HeadCfg.GEN.Torch_Mode = MODE_SINGLE_TORCH;

			// TVL
			m->pCfg->HeadCfg.SwitchHead.VECT_Indx = VECT_TVL;
			m->pCfg->HeadCfg.SwitchHead.TML_Indx = TML_AX_TVL;

			m->pCfg->HeadCfg.TVL.PROC_Indx = PROC_TVL;
			m->pCfg->HeadCfg.TVL.TML_Indx = TML_AX_TVL;

			// This is like BPV
			m->pCfg->HeadCfg.TVL.VECT_Indx = VECT_TVL;
			m->pCfg->HeadCfg.TVL.Enc_Dir = 1;

			//m->pCfg->HeadCfg.TVL.EncNominator = 39546 * 1024 * 4 / (1.875 * M_PI * 32 ) ;
			//m->pCfg->HeadCfg.TVL.EncDenominator = 540;
			//m->pCfg->HeadCfg.TVL.EncPerTick = (DINT)ceil(m->pCfg->HeadCfg.TVL.EncNominator / m->pCfg->HeadCfg.TVL.EncDenominator );

			m->pCfg->HeadCfg.TVL.EncScale = 540.0 *  (1.875 * M_PI * 32 ) / (39546 * 1024 * 4);
			m->pCfg->HeadCfg.TVL.EncPerTick = (DINT)ceil(1.0/m->pCfg->HeadCfg.TVL.EncScale);

			m->pCfg->HeadCfg.TVL.EncPerTick_SecEnc = 159; // (4000 * 4) / (1" * Pi * 32)
			m->pCfg->HeadCfg.TVL.PinsPerRot = 0;  // Dynamic Configuration
			m->pCfg->HeadCfg.TVL.DistPerTick = 25.4 /32.0; // 1/32"
			/////////////////////

			m->pCfg->HeadCfg.TVL.BtnJog_Gain = 24;
			m->pCfg->HeadCfg.TVL.BtnJog_Mode = BTN_JOG_MODE_SINGLE;

			// WF
			m->pCfg->HeadCfg.WF.PROC_Indx = PROC_WIRE_FEED;
			m->pCfg->HeadCfg.WF.VECT_A_Indx = VECT_WF;
			m->pCfg->HeadCfg.WF.VECT_B_Indx = VECT_WF_1;
			m->pCfg->HeadCfg.WF.TML_A_Indx = TML_AX_WF;
			m->pCfg->HeadCfg.WF.TML_B_Indx = TML_AX_WF_1;

			m->pCfg->HeadCfg.WF.VECT_Aux_A_Indx = VECT_AUX_WF;
			m->pCfg->HeadCfg.WF.VECT_Aux_B_Indx = VECT_AUX_WF_1;
			m->pCfg->HeadCfg.WF.TML_Aux_A_Indx = TML_AUX_AX_WF;
			m->pCfg->HeadCfg.WF.TML_Aux_B_Indx = TML_AUX_AX_WF_1;

			m->pCfg->HeadCfg.WF.BtnJog_Gain = 24;
			m->pCfg->HeadCfg.WF.BtnJog_Mode = BTN_JOG_MODE_SINGLE;

			// WP
			m->pCfg->HeadCfg.WP.PROC_Indx = PROC_WIRE_PULSE;
			m->pCfg->HeadCfg.WP.VECT_A_Indx = VECT_WP;
			m->pCfg->HeadCfg.WP.VECT_B_Indx = VECT_WP_1;
			m->pCfg->HeadCfg.WP.TML_A_Indx = TML_AX_WP;
			m->pCfg->HeadCfg.WP.TML_B_Indx = TML_AX_WP_1;

			// OSC
			m->pCfg->HeadCfg.OSC.PROC_Indx = PROC_OSC;
			m->pCfg->HeadCfg.OSC.VECT_A_Indx = VECT_OSC;
			m->pCfg->HeadCfg.OSC.VECT_B_Indx = VECT_OSC;
			m->pCfg->HeadCfg.OSC.TML_A_Indx = TML_AX_OSC;
			m->pCfg->HeadCfg.OSC.TML_B_Indx = TML_AX_OSC;
			m->pCfg->HeadCfg.OSC.Limits_Harcoded = 0;

			m->pCfg->HeadCfg.OSC.WhelJog_OnlyWhenRun = 0;

			m->pCfg->HeadCfg.OSC.BtnJog_Gain = 4;
			m->pCfg->HeadCfg.OSC.BtnJog_Mode = BTN_JOG_MODE_SINGLE;

			m->pCfg->HeadCfg.OSC.WheelJog_Gain1 = 0.2;
			m->pCfg->HeadCfg.OSC.WhelJog_Mode1 = WHL_JOG_MODE_STEP;

			m->pCfg->HeadCfg.OSC.WheelJog_Gain2 = 0.2;
			m->pCfg->HeadCfg.OSC.WhelJog_Mode2 = WHL_JOG_MODE_STEP;

			m->pCfg->HeadCfg.OSC.DwellDir = 1;

			// WRST
			m->pCfg->HeadCfg.WRST.PROC_Indx = PROC_WRST;
			m->pCfg->HeadCfg.WRST.VECT_A_Indx = VECT_WRST;
			m->pCfg->HeadCfg.WRST.VECT_B_Indx = VECT_WRST;
			m->pCfg->HeadCfg.WRST.TML_A_Indx = TML_AX_WRST;
			m->pCfg->HeadCfg.WRST.TML_B_Indx = TML_AX_WRST;
			m->pCfg->HeadCfg.WRST.Limits_Harcoded = 0;

			//m->pCfg->HeadCfg.WRST.BtnJog_Gain = 24.0;
			m->pCfg->HeadCfg.WRST.BtnJog_Gain = 0.24;
			m->pCfg->HeadCfg.WRST.BtnJog_Mode = BTN_JOG_MODE_SINGLE;

			// AVC
			m->pCfg->HeadCfg.AVC.PROC_Indx = PROC_AVC;
			m->pCfg->HeadCfg.AVC.VECT_A_Indx = VECT_AVC;
			m->pCfg->HeadCfg.AVC.VECT_B_Indx = VECT_AVC;
			m->pCfg->HeadCfg.AVC.TML_A_Indx = TML_AX_AVC;
			m->pCfg->HeadCfg.AVC.TML_B_Indx = TML_AX_AVC;

			m->pCfg->HeadCfg.AVC.BtnJog_Gain = 1;
			m->pCfg->HeadCfg.AVC.BtnJog_Mode = BTN_JOG_MODE_SINGLE;

			// INDX
			m->pCfg->HeadCfg.INDX.PROC_Indx = PROC_INDX;
			m->pCfg->HeadCfg.INDX.VECT_A_Indx = VECT_INDX_1;
			m->pCfg->HeadCfg.INDX.VECT_B_Indx = VECT_INDX_2;
			m->pCfg->HeadCfg.INDX.TML_A_Indx = TML_AX_INDX;
			m->pCfg->HeadCfg.INDX.TML_B_Indx = TML_AX_INDX_1;
			m->pCfg->HeadCfg.INDX.BtnJog_Gain = 1.0;

			// GAS
			m->pCfg->HeadCfg.GAS.PROC_Indx = PROC_GAS;

			// COOL
			m->pCfg->HeadCfg.COOL.PROC_Indx = PROC_COOL;

			// TIG
			m->pCfg->HeadCfg.TIG.PROC_Indx = PROC_TIG_PS;

			// HW
			m->pCfg->HeadCfg.HW.PROC_Indx = PROC_HW_PS;

			// WB
			m->pCfg->HeadCfg.WB[WB_UD].PROC_Indx = PROC_WB_UD;
			m->pCfg->HeadCfg.WB[WB_LR].PROC_Indx = PROC_WB_LR;

			m->pCfg->HeadCfg.WB[WB_UD].VECT_Indx = VECT_WB_UD;
			m->pCfg->HeadCfg.WB[WB_LR].VECT_Indx = VECT_WB_LR;

			// Lamp On Off
			m->pCfg->HeadCfg.LampOnOFF.VECT_A_Indx = VECT_OSC + 1;
			m->pCfg->HeadCfg.LampOnOFF.VECT_B_Indx = VECT_INDX_1 + 1;

			/////////////////////////////////////////////////////

			// frame size if zero always speed factor is 1.0
			//m->FrameDia = 4.5 * in_2_mm ;
			m->FrameDia = 0.0;

			switch(headType){

				case BPV_v2_MPBO:

					Configure_BPV_v2_MPBO(m , headType);
					DefaultCalibr_BPV_v2_MPBO(m->pDefaultCalib);

				break;

				case BPV_v2_MT:

					Configure_BPV_v2_MT(m , headType);
					DefaultCalibr_BPV_v2_MT(m->pDefaultCalib);

				break;

				case BPV_v2_MT_BO:

					Configure_BPV_v2_MT_BO(m , headType);
					DefaultCalibr_BPV_v2_MT_BO(m->pDefaultCalib);

				break;

			}

		break;

		/************ BPV_v2_MPGH - 17 ************/
		/************ BPV_v2_TT_BO_TOS - 21 ************/
		case BPV_v2_MPGH:
		case BPV_v2_TT_BO_TOS:

			m->pCfg->HeadCfg.GEN.Torch_Mode = MODE_SINGLE_TORCH;

			// TVL

			m->pCfg->HeadCfg.TVL.PROC_Indx = PROC_TVL;
			m->pCfg->HeadCfg.TVL.TML_Indx = TML_AX_TVL;

			// This is like BPV
			m->pCfg->HeadCfg.TVL.VECT_Indx = VECT_TVL;
			m->pCfg->HeadCfg.TVL.Enc_Dir = 1;

			//m->pCfg->HeadCfg.TVL.EncNominator = (75 * 50)  * 1024 * 4 / (0.625 * M_PI * 32 ) ;
			//m->pCfg->HeadCfg.TVL.EncDenominator = -19;
			//m->pCfg->HeadCfg.TVL.EncPerTick  = (DINT)ceil(m->pCfg->HeadCfg.TVL.EncNominator/m->pCfg->HeadCfg.TVL.EncDenominator);

			m->pCfg->HeadCfg.TVL.EncScale = -19.0 *  (0.625 * M_PI * 32 ) / ((75 * 50)  * 1024 * 4) ;
			m->pCfg->HeadCfg.TVL.EncPerTick = (DINT)ceil(1.0/m->pCfg->HeadCfg.TVL.EncScale);

			m->pCfg->HeadCfg.TVL.EncPerTick_SecEnc = 159; // (4000 * 4) / (1" * Pi * 32)
			m->pCfg->HeadCfg.TVL.PinsPerRot = 0;  // Dynamic Configuration
			m->pCfg->HeadCfg.TVL.DistPerTick = 25.4 /32.0; // 1/32"
			/////////////////////

			m->pCfg->HeadCfg.TVL.BtnJog_Gain = 24;
			m->pCfg->HeadCfg.TVL.BtnJog_Mode = BTN_JOG_MODE_SINGLE;

			// WF
			m->pCfg->HeadCfg.WF.PROC_Indx = PROC_WIRE_FEED;
			m->pCfg->HeadCfg.WF.VECT_A_Indx = VECT_WF;
			m->pCfg->HeadCfg.WF.VECT_B_Indx = VECT_WF;
			m->pCfg->HeadCfg.WF.TML_A_Indx = TML_AX_WF;
			m->pCfg->HeadCfg.WF.TML_B_Indx = TML_AX_WF;

			m->pCfg->HeadCfg.WF.BtnJog_Gain = 24;
			m->pCfg->HeadCfg.WF.BtnJog_Mode = BTN_JOG_MODE_SINGLE;

			// WP
			m->pCfg->HeadCfg.WP.PROC_Indx = PROC_WIRE_PULSE;
			m->pCfg->HeadCfg.WP.VECT_A_Indx = VECT_WP;
			m->pCfg->HeadCfg.WP.VECT_B_Indx = VECT_WP;
			m->pCfg->HeadCfg.WP.TML_A_Indx = TML_AX_WP;
			m->pCfg->HeadCfg.WP.TML_B_Indx = TML_AX_WP;

			// OSC
			m->pCfg->HeadCfg.OSC.PROC_Indx = PROC_OSC;
			m->pCfg->HeadCfg.OSC.VECT_A_Indx = VECT_OSC;
			m->pCfg->HeadCfg.OSC.VECT_B_Indx = VECT_OSC;
			m->pCfg->HeadCfg.OSC.TML_A_Indx = TML_AX_OSC;
			m->pCfg->HeadCfg.OSC.TML_B_Indx = TML_AX_OSC;
			m->pCfg->HeadCfg.OSC.Limits_Harcoded = 0;

			m->pCfg->HeadCfg.OSC.WhelJog_OnlyWhenRun = 0;

			m->pCfg->HeadCfg.OSC.BtnJog_Gain = 9;
			m->pCfg->HeadCfg.OSC.BtnJog_Mode = BTN_JOG_MODE_SINGLE;

			m->pCfg->HeadCfg.OSC.WheelJog_Gain1 = 0.2;
			m->pCfg->HeadCfg.OSC.WhelJog_Mode1 = WHL_JOG_MODE_STEP;

			m->pCfg->HeadCfg.OSC.WheelJog_Gain2 = 0.2;
			m->pCfg->HeadCfg.OSC.WhelJog_Mode2 = WHL_JOG_MODE_STEP;

			m->pCfg->HeadCfg.OSC.DwellDir = 1;

			// WRST
			m->pCfg->HeadCfg.WRST.PROC_Indx = PROC_WRST;
			m->pCfg->HeadCfg.WRST.VECT_A_Indx = VECT_WRST;
			m->pCfg->HeadCfg.WRST.VECT_B_Indx = VECT_WRST;
			m->pCfg->HeadCfg.WRST.TML_A_Indx = TML_AX_WRST;
			m->pCfg->HeadCfg.WRST.TML_B_Indx = TML_AX_WRST;
			m->pCfg->HeadCfg.WRST.Limits_Harcoded = 0;

			//m->pCfg->HeadCfg.WRST.BtnJog_Gain = 24.0;
			m->pCfg->HeadCfg.WRST.BtnJog_Gain = 0.24;
			m->pCfg->HeadCfg.WRST.BtnJog_Mode = BTN_JOG_MODE_SINGLE;

			// AVC
			m->pCfg->HeadCfg.AVC.PROC_Indx = PROC_AVC;
			m->pCfg->HeadCfg.AVC.VECT_A_Indx = VECT_AVC;
			m->pCfg->HeadCfg.AVC.VECT_B_Indx = VECT_AVC;
			m->pCfg->HeadCfg.AVC.TML_A_Indx = TML_AX_AVC;
			m->pCfg->HeadCfg.AVC.TML_B_Indx = TML_AX_AVC;

			m->pCfg->HeadCfg.AVC.BtnJog_Gain = 1;
			m->pCfg->HeadCfg.AVC.BtnJog_Mode = BTN_JOG_MODE_SINGLE;

			// INDX
			m->pCfg->HeadCfg.INDX.PROC_Indx = PROC_INDX;
			m->pCfg->HeadCfg.INDX.VECT_A_Indx = VECT_INDX_1;
			m->pCfg->HeadCfg.INDX.VECT_B_Indx = 0;
			m->pCfg->HeadCfg.INDX.TML_A_Indx = TML_AX_INDX;
			m->pCfg->HeadCfg.INDX.TML_B_Indx = 0;
			m->pCfg->HeadCfg.INDX.BtnJog_Gain = 1.0;

			// GAS
			m->pCfg->HeadCfg.GAS.PROC_Indx = PROC_GAS;

			// COOL
			m->pCfg->HeadCfg.COOL.PROC_Indx = PROC_COOL;

			// TIG
			m->pCfg->HeadCfg.TIG.PROC_Indx = PROC_TIG_PS;

			// HW
			m->pCfg->HeadCfg.HW.PROC_Indx = PROC_HW_PS;

			// WB
			m->pCfg->HeadCfg.WB[WB_UD].PROC_Indx = PROC_WB_UD;
			m->pCfg->HeadCfg.WB[WB_LR].PROC_Indx = PROC_WB_LR;

			m->pCfg->HeadCfg.WB[WB_UD].VECT_Indx = VECT_WB_UD;
			m->pCfg->HeadCfg.WB[WB_LR].VECT_Indx = VECT_WB_LR;

			// Lamp On Off

			m->pCfg->HeadCfg.LampOnOFF.VECT_A_Indx = 0;
			m->pCfg->HeadCfg.LampOnOFF.VECT_B_Indx = VECT_TVL;

			m->pCfg->HeadCfg.SwitchHead.VECT_Indx = VECT_INDX_1;
			m->pCfg->HeadCfg.SwitchHead.TML_Indx = TML_AX_INDX;

			/////////////////////////////////////////////////////

			// frame size if zero always speed factor is 1.0
			//m->FrameDia = 4.5 * in_2_mm ;
			m->FrameDia = 0.0;

			switch(headType){

				case BPV_v2_MPGH:

					Configure_BPV_v2_MPGH(m , headType);
					DefaultCalibr_BPV_v2_MPGH(m->pDefaultCalib);

				break;

				case BPV_v2_TT_BO_TOS:

					Configure_BPV_v2_TT_BO_TOS(m , headType);
					DefaultCalibr_BPV_v2_TT_BO_TOS(m->pDefaultCalib);

				break;

			}

		break;

		/************ BPV_v2_MPGV - 18 ************/
		/************ BPV_v2_MT_BO_TOS - 22 ************/
		case BPV_v2_MPGV:
		case BPV_v2_MT_BO_TOS:

			/////////

			m->pCfg->HeadCfg.GEN.Torch_Mode = MODE_SINGLE_TORCH;

			// TVL
			m->pCfg->HeadCfg.SwitchHead.VECT_Indx = VECT_TVL;
			m->pCfg->HeadCfg.SwitchHead.TML_Indx = TML_AX_TVL;

			m->pCfg->HeadCfg.TVL.PROC_Indx = PROC_TVL;
			m->pCfg->HeadCfg.TVL.TML_Indx = TML_AX_TVL;

			// This is like BPV
			m->pCfg->HeadCfg.TVL.VECT_Indx = VECT_TVL;
			m->pCfg->HeadCfg.TVL.Enc_Dir = 1;

			//m->pCfg->HeadCfg.TVL.EncNominator = 16209.6631 * 25.4;
			//m->pCfg->HeadCfg.TVL.EncDenominator = -32;
			//m->pCfg->HeadCfg.TVL.EncPerTick = (DINT)ceil(m->pCfg->HeadCfg.TVL.EncNominator / m->pCfg->HeadCfg.TVL.EncDenominator );

			m->pCfg->HeadCfg.TVL.EncScale = -32.0 /  (16209.6631 * 25.4);
			m->pCfg->HeadCfg.TVL.EncPerTick = (DINT)ceil(1.0/m->pCfg->HeadCfg.TVL.EncScale);

			m->pCfg->HeadCfg.TVL.EncPerTick_SecEnc = 159; // (4000 * 4) / (1" * Pi * 32)
			m->pCfg->HeadCfg.TVL.PinsPerRot = 0;  // Dynamic Configuration
			m->pCfg->HeadCfg.TVL.DistPerTick = 25.4 /32.0; // 1/32"
			/////////////////////

			m->pCfg->HeadCfg.TVL.BtnJog_Gain = 24;
			m->pCfg->HeadCfg.TVL.BtnJog_Mode = BTN_JOG_MODE_SINGLE;

			// WF
			m->pCfg->HeadCfg.WF.PROC_Indx = PROC_WIRE_FEED;
			m->pCfg->HeadCfg.WF.VECT_A_Indx = VECT_WF;
			m->pCfg->HeadCfg.WF.VECT_B_Indx = VECT_WF_1;
			m->pCfg->HeadCfg.WF.TML_A_Indx = TML_AX_WF;
			m->pCfg->HeadCfg.WF.TML_B_Indx = TML_AX_WF_1;

			m->pCfg->HeadCfg.WF.VECT_Aux_A_Indx = VECT_AUX_WF;
			m->pCfg->HeadCfg.WF.VECT_Aux_B_Indx = VECT_AUX_WF_1;
			m->pCfg->HeadCfg.WF.TML_Aux_A_Indx = TML_AUX_AX_WF;
			m->pCfg->HeadCfg.WF.TML_Aux_B_Indx = TML_AUX_AX_WF_1;

			m->pCfg->HeadCfg.WF.BtnJog_Gain = 24;
			m->pCfg->HeadCfg.WF.BtnJog_Mode = BTN_JOG_MODE_SINGLE;

			// WP
			m->pCfg->HeadCfg.WP.PROC_Indx = PROC_WIRE_PULSE;
			m->pCfg->HeadCfg.WP.VECT_A_Indx = VECT_WP;
			m->pCfg->HeadCfg.WP.VECT_B_Indx = VECT_WP_1;
			m->pCfg->HeadCfg.WP.TML_A_Indx = TML_AX_WP;
			m->pCfg->HeadCfg.WP.TML_B_Indx = TML_AX_WP_1;

			// OSC
			m->pCfg->HeadCfg.OSC.PROC_Indx = PROC_OSC;
			m->pCfg->HeadCfg.OSC.VECT_A_Indx = VECT_OSC;
			m->pCfg->HeadCfg.OSC.VECT_B_Indx = VECT_OSC;
			m->pCfg->HeadCfg.OSC.TML_A_Indx = TML_AX_OSC;
			m->pCfg->HeadCfg.OSC.TML_B_Indx = TML_AX_OSC;
			m->pCfg->HeadCfg.OSC.Limits_Harcoded = 0;

			m->pCfg->HeadCfg.OSC.WhelJog_OnlyWhenRun = 0;

			m->pCfg->HeadCfg.OSC.BtnJog_Gain = 17;
			m->pCfg->HeadCfg.OSC.BtnJog_Mode = BTN_JOG_MODE_SINGLE;

			m->pCfg->HeadCfg.OSC.WheelJog_Gain1 = 0.2;
			m->pCfg->HeadCfg.OSC.WhelJog_Mode1 = WHL_JOG_MODE_STEP;

			m->pCfg->HeadCfg.OSC.WheelJog_Gain2 = 0.2;
			m->pCfg->HeadCfg.OSC.WhelJog_Mode2 = WHL_JOG_MODE_STEP;

			m->pCfg->HeadCfg.OSC.DwellDir = 1;

			// WRST
			m->pCfg->HeadCfg.WRST.PROC_Indx = PROC_WRST;
			m->pCfg->HeadCfg.WRST.VECT_A_Indx = VECT_WRST;
			m->pCfg->HeadCfg.WRST.VECT_B_Indx = VECT_WRST;
			m->pCfg->HeadCfg.WRST.TML_A_Indx = TML_AX_WRST;
			m->pCfg->HeadCfg.WRST.TML_B_Indx = TML_AX_WRST;
			m->pCfg->HeadCfg.WRST.Limits_Harcoded = 0;

			//m->pCfg->HeadCfg.WRST.BtnJog_Gain = 24.0;
			m->pCfg->HeadCfg.WRST.BtnJog_Gain = 0.24;
			m->pCfg->HeadCfg.WRST.BtnJog_Mode = BTN_JOG_MODE_SINGLE;

			// AVC
			m->pCfg->HeadCfg.AVC.PROC_Indx = PROC_AVC;
			m->pCfg->HeadCfg.AVC.VECT_A_Indx = VECT_AVC;
			m->pCfg->HeadCfg.AVC.VECT_B_Indx = VECT_AVC;
			m->pCfg->HeadCfg.AVC.TML_A_Indx = TML_AX_AVC;
			m->pCfg->HeadCfg.AVC.TML_B_Indx = TML_AX_AVC;

			m->pCfg->HeadCfg.AVC.BtnJog_Gain = 1;
			m->pCfg->HeadCfg.AVC.BtnJog_Mode = BTN_JOG_MODE_SINGLE;

			// INDX

			m->pCfg->HeadCfg.INDX.PROC_Indx = PROC_INDX;
			m->pCfg->HeadCfg.INDX.VECT_A_Indx = VECT_INDX_1;
			m->pCfg->HeadCfg.INDX.VECT_B_Indx = VECT_INDX_2;
			m->pCfg->HeadCfg.INDX.TML_A_Indx = TML_AX_INDX;
			m->pCfg->HeadCfg.INDX.TML_B_Indx = TML_AX_INDX_1;
			m->pCfg->HeadCfg.INDX.BtnJog_Gain = 1.0;

			// GAS
			m->pCfg->HeadCfg.GAS.PROC_Indx = PROC_GAS;

			// COOL
			m->pCfg->HeadCfg.COOL.PROC_Indx = PROC_COOL;

			// TIG
			m->pCfg->HeadCfg.TIG.PROC_Indx = PROC_TIG_PS;

			// HW
			m->pCfg->HeadCfg.HW.PROC_Indx = PROC_HW_PS;

			// WB
			m->pCfg->HeadCfg.WB[WB_UD].PROC_Indx = PROC_WB_UD;
			m->pCfg->HeadCfg.WB[WB_LR].PROC_Indx = PROC_WB_LR;

			m->pCfg->HeadCfg.WB[WB_UD].VECT_Indx = VECT_WB_UD;
			m->pCfg->HeadCfg.WB[WB_LR].VECT_Indx = VECT_WB_LR;

			// Lamp On Off
			m->pCfg->HeadCfg.LampOnOFF.VECT_A_Indx = VECT_OSC + 1;
			m->pCfg->HeadCfg.LampOnOFF.VECT_B_Indx = VECT_INDX_1 + 1;

			/////////////////////////////////////////////////////

			// frame size if zero always speed factor is 1.0
			//m->FrameDia = 4.5 * in_2_mm ;
			m->FrameDia = 0.0;

			switch(headType){

				case BPV_v2_MPGV:

					Configure_BPV_v2_MPGV(m , headType);
					DefaultCalibr_BPV_v2_MPGV(m->pDefaultCalib);

				break;

				case BPV_v2_MT_BO_TOS:

					Configure_BPV_v2_MT_BO_TOS(m , headType);
					DefaultCalibr_BPV_v2_MT_BO_TOS(m->pDefaultCalib);

				break;

			}

		break;

		///////////////////////////////////////////////////////////////////////////////

		/************ 23 ************/
		case RUBIX:

			m->pCfg->HeadCfg.GEN.Torch_Mode = MODE_SINGLE_TORCH;

			// TVL
			m->pCfg->HeadCfg.SwitchHead.VECT_Indx = 0;
			m->pCfg->HeadCfg.SwitchHead.TML_Indx = 0;

			m->pCfg->HeadCfg.TVL.PROC_Indx = PROC_TVL;
			m->pCfg->HeadCfg.TVL.TML_Indx = TML_AX_TVL;
			m->pCfg->HeadCfg.TVL.DC_Indx = 0;

			m->pCfg->HeadCfg.TVL.VECT_Indx = VECT_TVL;
			m->pCfg->HeadCfg.TVL.Enc_Dir = 1;
			m->pCfg->HeadCfg.TVL.EncPerTick = 38;  // 1/16 inch
			m->pCfg->HeadCfg.TVL.PinsPerRot = 0;  // Dynamic Configuration
			m->pCfg->HeadCfg.TVL.DistPerTick = 25.4 /16.0; // 1/16"

			m->pCfg->HeadCfg.TVL.BtnJog_Gain = 24;
			m->pCfg->HeadCfg.TVL.BtnJog_Mode = BTN_JOG_MODE_SINGLE;

			// WF
			m->pCfg->HeadCfg.WF.PROC_Indx = PROC_WIRE_FEED;
			m->pCfg->HeadCfg.WF.VECT_A_Indx = VECT_WF;
			m->pCfg->HeadCfg.WF.VECT_B_Indx = VECT_WF;
			m->pCfg->HeadCfg.WF.TML_A_Indx = TML_AX_WF;
			m->pCfg->HeadCfg.WF.TML_B_Indx = TML_AX_WF;
			//m->pCfg->HeadCfg.WF.DC_A_Indx = DC_AX_WF;
			//m->pCfg->HeadCfg.WF.DC_B_Indx = DC_AX_WF;

			m->pCfg->HeadCfg.WF.BtnJog_Gain = 24;
			m->pCfg->HeadCfg.WF.BtnJog_Mode = BTN_JOG_MODE_SINGLE;

			// WP
			m->pCfg->HeadCfg.WP.PROC_Indx = PROC_WIRE_PULSE;
			m->pCfg->HeadCfg.WP.VECT_A_Indx = 0;
			m->pCfg->HeadCfg.WP.VECT_B_Indx = 0;
			/*
			m->pCfg->HeadCfg.WP.VECT_A_Indx = VECT_WP;
			m->pCfg->HeadCfg.WP.VECT_B_Indx = VECT_WP;
			m->pCfg->HeadCfg.WP.DC_A_Indx = DC_AX_WP;
			m->pCfg->HeadCfg.WP.DC_B_Indx = DC_AX_WP;
			*/

			// OSC
			m->pCfg->HeadCfg.OSC.PROC_Indx = PROC_OSC;
			m->pCfg->HeadCfg.OSC.VECT_A_Indx = VECT_OSC;
			m->pCfg->HeadCfg.OSC.VECT_B_Indx = VECT_OSC;
			m->pCfg->HeadCfg.OSC.TML_A_Indx = TML_AX_OSC;
			m->pCfg->HeadCfg.OSC.TML_B_Indx = TML_AX_OSC;
			m->pCfg->HeadCfg.OSC.Limits_Harcoded = 0;

			m->pCfg->HeadCfg.OSC.BtnJog_Gain = 24.0;
			m->pCfg->HeadCfg.OSC.BtnJog_Mode = BTN_JOG_MODE_SINGLE;

			m->pCfg->HeadCfg.OSC.WheelJog_Gain1 = 5;
			m->pCfg->HeadCfg.OSC.WhelJog_Mode1 = WHL_JOG_MODE_STEP;

			m->pCfg->HeadCfg.OSC.WheelJog_Gain2 = 0.2;
			m->pCfg->HeadCfg.OSC.WhelJog_Mode2 = WHL_JOG_MODE_STEP;
			m->pCfg->HeadCfg.OSC.WhelJog_OnlyWhenRun = 1;

			m->pCfg->HeadCfg.OSC.DwellDir = 1;

			// AVC
			m->pCfg->HeadCfg.AVC.PROC_Indx = PROC_AVC;
			m->pCfg->HeadCfg.AVC.VECT_A_Indx = VECT_AVC;
			m->pCfg->HeadCfg.AVC.VECT_B_Indx = VECT_AVC;
			m->pCfg->HeadCfg.AVC.TML_A_Indx = TML_AX_AVC;
			m->pCfg->HeadCfg.AVC.TML_B_Indx = TML_AX_AVC;

			m->pCfg->HeadCfg.AVC.BtnJog_Gain = 24;
			m->pCfg->HeadCfg.AVC.BtnJog_Mode = BTN_JOG_MODE_SINGLE;

			// GAS
			m->pCfg->HeadCfg.GAS.PROC_Indx = PROC_GAS;

			// COOL
			m->pCfg->HeadCfg.COOL.PROC_Indx = PROC_COOL;

			// TIG
			m->pCfg->HeadCfg.TIG.PROC_Indx = PROC_TIG_PS;

			// HW
			m->pCfg->HeadCfg.HW.PROC_Indx = PROC_HW_PS;

			// INDX
			m->pCfg->HeadCfg.INDX.PROC_Indx = PROC_INDX; // Must be even is disabled

			// WB
			m->pCfg->HeadCfg.WB[WB_UD].PROC_Indx = PROC_WB_UD;
			m->pCfg->HeadCfg.WB[WB_LR].PROC_Indx = PROC_WB_LR;

			m->pCfg->HeadCfg.WB[WB_UD].VECT_Indx = VECT_WB_UD;
			m->pCfg->HeadCfg.WB[WB_LR].VECT_Indx = VECT_WB_LR;

			// Lamp On Off
			m->pCfg->HeadCfg.LampOnOFF.VECT_A_Indx = 0; // 0 - not used
			m->pCfg->HeadCfg.LampOnOFF.VECT_B_Indx = 0; // 0 - not used

			//////////////////////
			// frame size if zero always speed factor is 1.0
			//m->FrameDia = 4.5 * in_2_mm ;
			m->FrameDia = 0.0;

			Configure_RUBIX(m , RUBIX);
			DefaultCalibr_RUBIX(m->pDefaultCalib);

		break;

		///////////////////////////////////////////////////////////////////////////////

		/************ 24 ************/
		case F_HEAD_MINI_STND:

			m->pCfg->HeadCfg.GEN.Torch_Mode = MODE_SINGLE_TORCH;

			// TVL
			m->pCfg->HeadCfg.SwitchHead.VECT_Indx = 0;
			m->pCfg->HeadCfg.SwitchHead.TML_Indx = 0;

			m->pCfg->HeadCfg.TVL.PROC_Indx = PROC_TVL;
			m->pCfg->HeadCfg.TVL.TML_Indx = TML_AX_TVL;
			m->pCfg->HeadCfg.TVL.DC_Indx = 0;

			m->pCfg->HeadCfg.TVL.VECT_Indx = VECT_TVL;
			m->pCfg->HeadCfg.TVL.Enc_Dir = 1;
			m->pCfg->HeadCfg.TVL.EncPerTick = 38;  // 1/16 inch
			m->pCfg->HeadCfg.TVL.PinsPerRot = 0;  // Dynamic Configuration
			m->pCfg->HeadCfg.TVL.DistPerTick = 25.4 /16.0; // 1/16"

			m->pCfg->HeadCfg.TVL.BtnJog_Gain = 24;
			m->pCfg->HeadCfg.TVL.BtnJog_Mode = BTN_JOG_MODE_SINGLE;

			// WF
			m->pCfg->HeadCfg.WF.PROC_Indx = PROC_WIRE_FEED;
			m->pCfg->HeadCfg.WF.VECT_A_Indx = VECT_WF;
			m->pCfg->HeadCfg.WF.VECT_B_Indx = VECT_WF;
			m->pCfg->HeadCfg.WF.TML_A_Indx = TML_AX_WF;
			m->pCfg->HeadCfg.WF.TML_B_Indx = TML_AX_WF;

			m->pCfg->HeadCfg.WF.BtnJog_Gain = 24;
			m->pCfg->HeadCfg.WF.BtnJog_Mode = BTN_JOG_MODE_SINGLE;

			// WP
			m->pCfg->HeadCfg.WP.PROC_Indx = PROC_WIRE_PULSE;
			m->pCfg->HeadCfg.WP.VECT_A_Indx = 0;
			m->pCfg->HeadCfg.WP.VECT_B_Indx = 0;

			// OSC
			m->pCfg->HeadCfg.OSC.PROC_Indx = PROC_OSC;
			m->pCfg->HeadCfg.OSC.VECT_A_Indx = VECT_OSC;
			m->pCfg->HeadCfg.OSC.VECT_B_Indx = VECT_OSC;
			m->pCfg->HeadCfg.OSC.TML_A_Indx = TML_AX_OSC;
			m->pCfg->HeadCfg.OSC.TML_B_Indx = TML_AX_OSC;
			m->pCfg->HeadCfg.OSC.Limits_Harcoded = 0;

			m->pCfg->HeadCfg.OSC.BtnJog_Gain = 24.0;
			m->pCfg->HeadCfg.OSC.BtnJog_Mode = BTN_JOG_MODE_SINGLE;

			m->pCfg->HeadCfg.OSC.WheelJog_Gain1 = 5;
			m->pCfg->HeadCfg.OSC.WhelJog_Mode1 = WHL_JOG_MODE_STEP;

			m->pCfg->HeadCfg.OSC.WheelJog_Gain2 = 0.2;
			m->pCfg->HeadCfg.OSC.WhelJog_Mode2 = WHL_JOG_MODE_STEP;
			m->pCfg->HeadCfg.OSC.WhelJog_OnlyWhenRun = 1;

			m->pCfg->HeadCfg.OSC.DwellDir = 1;

			// AVC
			m->pCfg->HeadCfg.AVC.PROC_Indx = PROC_AVC;
			m->pCfg->HeadCfg.AVC.VECT_A_Indx = VECT_AVC;
			m->pCfg->HeadCfg.AVC.VECT_B_Indx = VECT_AVC;
			m->pCfg->HeadCfg.AVC.TML_A_Indx = TML_AX_AVC;
			m->pCfg->HeadCfg.AVC.TML_B_Indx = TML_AX_AVC;

			m->pCfg->HeadCfg.AVC.BtnJog_Gain = 24;
			m->pCfg->HeadCfg.AVC.BtnJog_Mode = BTN_JOG_MODE_SINGLE;

			// GAS
			m->pCfg->HeadCfg.GAS.PROC_Indx = PROC_GAS;

			// COOL
			m->pCfg->HeadCfg.COOL.PROC_Indx = PROC_COOL;

			// TIG
			m->pCfg->HeadCfg.TIG.PROC_Indx = PROC_TIG_PS;

			// HW
			m->pCfg->HeadCfg.HW.PROC_Indx = PROC_HW_PS;

			// INDX
			m->pCfg->HeadCfg.INDX.PROC_Indx = PROC_INDX; // Must be even is disabled

			// WB
			m->pCfg->HeadCfg.WB[WB_UD].PROC_Indx = PROC_WB_UD;
			m->pCfg->HeadCfg.WB[WB_LR].PROC_Indx = PROC_WB_LR;

			m->pCfg->HeadCfg.WB[WB_UD].VECT_Indx = VECT_WB_UD;
			m->pCfg->HeadCfg.WB[WB_LR].VECT_Indx = VECT_WB_LR;

			// Lamp On Off
			m->pCfg->HeadCfg.LampOnOFF.VECT_A_Indx = 0; // 0 - not used
			m->pCfg->HeadCfg.LampOnOFF.VECT_B_Indx = 0; // 0 - not used

			//////////////////////
			// frame size if zero always speed factor is 1.0
			//m->FrameDia = 4.5 * in_2_mm ;
			m->FrameDia = 0.0;

			Configure_F_HEAD_MINI_STND(m , F_HEAD_MINI_STND);
			DefaultCalibr_F_HEAD_MINI_STND(m->pDefaultCalib);

		break;

		/************ 25 ************/
		case F_HEAD_MINI_OMEGA: 		// Like F_HEAD_HP_MINI_ENC [7]

			m->pCfg->HeadCfg.GEN.Torch_Mode = MODE_SINGLE_TORCH;

			// TVL
			m->pCfg->HeadCfg.SwitchHead.VECT_Indx = 0;
			m->pCfg->HeadCfg.SwitchHead.TML_Indx = 0;

			m->pCfg->HeadCfg.TVL.PROC_Indx = PROC_TVL;
			m->pCfg->HeadCfg.TVL.TML_Indx = TML_AX_TVL;
			m->pCfg->HeadCfg.TVL.DC_Indx = 0;

			m->pCfg->HeadCfg.TVL.VECT_Indx = VECT_TVL;
			m->pCfg->HeadCfg.TVL.Enc_Dir = 1;
			m->pCfg->HeadCfg.TVL.EncPerTick = 38;  // 1/16 inch
			m->pCfg->HeadCfg.TVL.PinsPerRot = 0;  // Dynamic Configuration
			m->pCfg->HeadCfg.TVL.DistPerTick = 25.4 /16.0; // 1/16"

			m->pCfg->HeadCfg.TVL.BtnJog_Gain = 24;
			m->pCfg->HeadCfg.TVL.BtnJog_Mode = BTN_JOG_MODE_SINGLE;

			// WF
			m->pCfg->HeadCfg.WF.PROC_Indx = PROC_WIRE_FEED;
			m->pCfg->HeadCfg.WF.VECT_A_Indx = VECT_WF;
			m->pCfg->HeadCfg.WF.VECT_B_Indx = VECT_WF;
			m->pCfg->HeadCfg.WF.DC_A_Indx = DC_AX_WF;
			m->pCfg->HeadCfg.WF.DC_B_Indx = DC_AX_WF;

			m->pCfg->HeadCfg.WF.BtnJog_Gain = 24;
			m->pCfg->HeadCfg.WF.BtnJog_Mode = BTN_JOG_MODE_SINGLE;

			// WP
			m->pCfg->HeadCfg.WP.PROC_Indx = PROC_WIRE_PULSE;
			m->pCfg->HeadCfg.WP.VECT_A_Indx = VECT_WP;
			m->pCfg->HeadCfg.WP.VECT_B_Indx = VECT_WP;
			m->pCfg->HeadCfg.WP.DC_A_Indx = DC_AX_WP;
			m->pCfg->HeadCfg.WP.DC_B_Indx = DC_AX_WP;

			// OSC
			m->pCfg->HeadCfg.OSC.PROC_Indx = PROC_OSC;
			m->pCfg->HeadCfg.OSC.VECT_A_Indx = VECT_OSC;
			m->pCfg->HeadCfg.OSC.VECT_B_Indx = VECT_OSC;
			m->pCfg->HeadCfg.OSC.TML_A_Indx = TML_AX_OSC;
			m->pCfg->HeadCfg.OSC.TML_B_Indx = TML_AX_OSC;
			m->pCfg->HeadCfg.OSC.Limits_Harcoded = 0;

			m->pCfg->HeadCfg.OSC.BtnJog_Gain = 24.0;
			m->pCfg->HeadCfg.OSC.BtnJog_Mode = BTN_JOG_MODE_SINGLE;

			m->pCfg->HeadCfg.OSC.WheelJog_Gain1 = 5;
			m->pCfg->HeadCfg.OSC.WhelJog_Mode1 = WHL_JOG_MODE_STEP;

			m->pCfg->HeadCfg.OSC.WheelJog_Gain2 = 0.2;
			m->pCfg->HeadCfg.OSC.WhelJog_Mode2 = WHL_JOG_MODE_STEP;
			m->pCfg->HeadCfg.OSC.WhelJog_OnlyWhenRun = 1;

			m->pCfg->HeadCfg.OSC.DwellDir = 1;

			// AVC
			m->pCfg->HeadCfg.AVC.PROC_Indx = PROC_AVC;
			m->pCfg->HeadCfg.AVC.VECT_A_Indx = VECT_AVC;
			m->pCfg->HeadCfg.AVC.VECT_B_Indx = VECT_AVC;
			m->pCfg->HeadCfg.AVC.TML_A_Indx = TML_AX_AVC;
			m->pCfg->HeadCfg.AVC.TML_B_Indx = TML_AX_AVC;

			m->pCfg->HeadCfg.AVC.BtnJog_Gain = 24;
			m->pCfg->HeadCfg.AVC.BtnJog_Mode = BTN_JOG_MODE_SINGLE;

			// GAS
			m->pCfg->HeadCfg.GAS.PROC_Indx = PROC_GAS;

			// COOL
			m->pCfg->HeadCfg.COOL.PROC_Indx = PROC_COOL;

			// TIG
			m->pCfg->HeadCfg.TIG.PROC_Indx = PROC_TIG_PS;

			// HW
			m->pCfg->HeadCfg.HW.PROC_Indx = PROC_HW_PS;

			// INDX
			m->pCfg->HeadCfg.INDX.PROC_Indx = PROC_INDX; // Must be even is disabled

			// WB
			m->pCfg->HeadCfg.WB[WB_UD].PROC_Indx = PROC_WB_UD;
			m->pCfg->HeadCfg.WB[WB_LR].PROC_Indx = PROC_WB_LR;

			m->pCfg->HeadCfg.WB[WB_UD].VECT_Indx = VECT_WB_UD;
			m->pCfg->HeadCfg.WB[WB_LR].VECT_Indx = VECT_WB_LR;

			// Lamp On Off
			m->pCfg->HeadCfg.LampOnOFF.VECT_A_Indx = 0; // 0 - not used
			m->pCfg->HeadCfg.LampOnOFF.VECT_B_Indx = 0; // 0 - not used

			//////////////////////
			// frame size if zero always speed factor is 1.0
			//m->FrameDia = 4.5 * in_2_mm ;
			m->FrameDia = 0.0;

			Configure_F_HEAD_MINI_OMEGA(m , F_HEAD_MINI_OMEGA);
			DefaultCalibr_F_HEAD_MINI_OMEGA(m->pDefaultCalib);

		break;

		/************ 26 ************/
		case D_HEAD_HP: 		// Like F_HEAD_MINI_OMEGA [25]	????

			m->pCfg->HeadCfg.GEN.Torch_Mode = MODE_SINGLE_TORCH;

			// TVL
			m->pCfg->HeadCfg.SwitchHead.VECT_Indx = 0;
			m->pCfg->HeadCfg.SwitchHead.TML_Indx = 0;

			m->pCfg->HeadCfg.TVL.PROC_Indx = PROC_TVL;
			m->pCfg->HeadCfg.TVL.TML_Indx = TML_AX_TVL;
			m->pCfg->HeadCfg.TVL.DC_Indx = 0;

			m->pCfg->HeadCfg.TVL.VECT_Indx = VECT_TVL;
			m->pCfg->HeadCfg.TVL.Enc_Dir = 1;
			m->pCfg->HeadCfg.TVL.EncPerTick = 38;  // 1/16 inch
			m->pCfg->HeadCfg.TVL.PinsPerRot = 0;  // Dynamic Configuration
			m->pCfg->HeadCfg.TVL.DistPerTick = 25.4 /16.0; // 1/16"

			m->pCfg->HeadCfg.TVL.BtnJog_Gain = 24;
			m->pCfg->HeadCfg.TVL.BtnJog_Mode = BTN_JOG_MODE_SINGLE;

			// WF
			m->pCfg->HeadCfg.WF.PROC_Indx = PROC_WIRE_FEED;
			m->pCfg->HeadCfg.WF.VECT_A_Indx = VECT_WF;
			m->pCfg->HeadCfg.WF.VECT_B_Indx = VECT_WF;
			m->pCfg->HeadCfg.WF.DC_A_Indx = DC_AX_WF;
			m->pCfg->HeadCfg.WF.DC_B_Indx = DC_AX_WF;

			m->pCfg->HeadCfg.WF.BtnJog_Gain = 24;
			m->pCfg->HeadCfg.WF.BtnJog_Mode = BTN_JOG_MODE_SINGLE;

			// WP
			m->pCfg->HeadCfg.WP.PROC_Indx = PROC_WIRE_PULSE;
			m->pCfg->HeadCfg.WP.VECT_A_Indx = VECT_WP;
			m->pCfg->HeadCfg.WP.VECT_B_Indx = VECT_WP;
			m->pCfg->HeadCfg.WP.DC_A_Indx = DC_AX_WP;
			m->pCfg->HeadCfg.WP.DC_B_Indx = DC_AX_WP;

			// OSC
			m->pCfg->HeadCfg.OSC.PROC_Indx = PROC_OSC;
			m->pCfg->HeadCfg.OSC.VECT_A_Indx = VECT_OSC;
			m->pCfg->HeadCfg.OSC.VECT_B_Indx = VECT_OSC;
			m->pCfg->HeadCfg.OSC.TML_A_Indx = TML_AX_OSC;
			m->pCfg->HeadCfg.OSC.TML_B_Indx = TML_AX_OSC;
			m->pCfg->HeadCfg.OSC.Limits_Harcoded = 0;

			m->pCfg->HeadCfg.OSC.BtnJog_Gain = 24.0;
			m->pCfg->HeadCfg.OSC.BtnJog_Mode = BTN_JOG_MODE_SINGLE;

			m->pCfg->HeadCfg.OSC.WheelJog_Gain1 = 5;
			m->pCfg->HeadCfg.OSC.WhelJog_Mode1 = WHL_JOG_MODE_STEP;

			m->pCfg->HeadCfg.OSC.WheelJog_Gain2 = 0.2;
			m->pCfg->HeadCfg.OSC.WhelJog_Mode2 = WHL_JOG_MODE_STEP;
			m->pCfg->HeadCfg.OSC.WhelJog_OnlyWhenRun = 1;

			m->pCfg->HeadCfg.OSC.DwellDir = 1;

			// AVC
			m->pCfg->HeadCfg.AVC.PROC_Indx = PROC_AVC;
			m->pCfg->HeadCfg.AVC.VECT_A_Indx = VECT_AVC;
			m->pCfg->HeadCfg.AVC.VECT_B_Indx = VECT_AVC;
			m->pCfg->HeadCfg.AVC.TML_A_Indx = TML_AX_AVC;
			m->pCfg->HeadCfg.AVC.TML_B_Indx = TML_AX_AVC;

			m->pCfg->HeadCfg.AVC.BtnJog_Gain = 24;
			m->pCfg->HeadCfg.AVC.BtnJog_Mode = BTN_JOG_MODE_SINGLE;

			// GAS
			m->pCfg->HeadCfg.GAS.PROC_Indx = PROC_GAS;

			// COOL
			m->pCfg->HeadCfg.COOL.PROC_Indx = PROC_COOL;

			// TIG
			m->pCfg->HeadCfg.TIG.PROC_Indx = PROC_TIG_PS;

			// HW
			m->pCfg->HeadCfg.HW.PROC_Indx = PROC_HW_PS;

			// INDX
			m->pCfg->HeadCfg.INDX.PROC_Indx = PROC_INDX; // Must be even is disabled

			// WB
			m->pCfg->HeadCfg.WB[WB_UD].PROC_Indx = PROC_WB_UD;
			m->pCfg->HeadCfg.WB[WB_LR].PROC_Indx = PROC_WB_LR;

			m->pCfg->HeadCfg.WB[WB_UD].VECT_Indx = VECT_WB_UD;
			m->pCfg->HeadCfg.WB[WB_LR].VECT_Indx = VECT_WB_LR;

			// Lamp On Off
			m->pCfg->HeadCfg.LampOnOFF.VECT_A_Indx = 0; // 0 - not used
			m->pCfg->HeadCfg.LampOnOFF.VECT_B_Indx = 0; // 0 - not used

			//////////////////////
			// frame size if zero always speed factor is 1.0
			//m->FrameDia = 4.5 * in_2_mm ;
			m->FrameDia = 0.0;

			Configure_D_HEAD_HP(m , D_HEAD_HP);
			DefaultCalibr_D_HEAD_HP(m->pDefaultCalib);

		break;

		/************ 31 ************/
		case CLAMSHELL_HEAD: // Based on BPV_F_HEAD

			m->pCfg->HeadCfg.GEN.Torch_Mode = MODE_SINGLE_TORCH;
			m->pCfg->HeadCfg.GEN.AVC_Mode = MODE_DUAL_AVC;

			// Gas SOlenoid & WRST
			/*
			m->pCfg->HeadCfg.SwitchHead.VECT_Indx = TML_AX_WRST + 1;
			m->pCfg->HeadCfg.SwitchHead.TML_Indx = TML_AX_WF_1 + 1;
			*/

			/** WF & WP -
			m->pCfg->HeadCfg.SwitchHead.VECT_Indx_2 = VECT_WF + 1;
			m->pCfg->HeadCfg.SwitchHead.TML_Indx_2 = TML_AX_WF + 1;
			*/

			//////
			m->pCfg->HeadCfg.TVL.PROC_Indx = PROC_TVL;
			m->pCfg->HeadCfg.TVL.TML_Indx = TML_AX_TVL;

			m->pCfg->HeadCfg.TVL.VECT_Indx = VECT_TVL;
			m->pCfg->HeadCfg.TVL.Enc_Dir = 1;
			//m->pCfg->HeadCfg.TVL.EncPerTick  = 5085;  //  5084.8094458543457034129135792358	// For 1/32 "
			m->pCfg->HeadCfg.TVL.EncPerTick  = 9800; // aby bylo 32 razy
			m->pCfg->HeadCfg.TVL.EncPerTick_SecEnc = 159; // (4000 * 4) / (1" * Pi * 32)
			m->pCfg->HeadCfg.TVL.PinsPerRot = 0;  // Dynamic Configuration
			m->pCfg->HeadCfg.TVL.DistPerTick = 25.4 /32.0; // 1/32"

			m->pCfg->HeadCfg.TVL.BtnJog_Gain = 24;
			m->pCfg->HeadCfg.TVL.BtnJog_Mode = BTN_JOG_MODE_SINGLE;

			// WF
			m->pCfg->HeadCfg.WF.PROC_Indx = PROC_WIRE_FEED;
			m->pCfg->HeadCfg.WF.VECT_A_Indx = VECT_WF;
			m->pCfg->HeadCfg.WF.VECT_B_Indx = VECT_WF;
			m->pCfg->HeadCfg.WF.TML_A_Indx = TML_AX_WF;
			m->pCfg->HeadCfg.WF.TML_B_Indx = TML_AX_WF;

			m->pCfg->HeadCfg.WF.BtnJog_Gain = 24;
			m->pCfg->HeadCfg.WF.BtnJog_Mode = BTN_JOG_MODE_SINGLE;

			// WP
			m->pCfg->HeadCfg.WP.PROC_Indx = PROC_WIRE_PULSE;
			m->pCfg->HeadCfg.WP.VECT_A_Indx = VECT_WP;
			m->pCfg->HeadCfg.WP.VECT_B_Indx = VECT_WP;
			m->pCfg->HeadCfg.WP.TML_A_Indx = TML_AX_WP;
			m->pCfg->HeadCfg.WP.TML_B_Indx = TML_AX_WP;

			// OSC
			m->pCfg->HeadCfg.OSC.PROC_Indx = PROC_OSC;
			m->pCfg->HeadCfg.OSC.VECT_A_Indx = VECT_OSC;
			m->pCfg->HeadCfg.OSC.VECT_B_Indx = VECT_OSC;
			m->pCfg->HeadCfg.OSC.TML_A_Indx = TML_AX_OSC;
			m->pCfg->HeadCfg.OSC.TML_B_Indx = TML_AX_OSC;
			m->pCfg->HeadCfg.OSC.Limits_Harcoded = 0;

			m->pCfg->HeadCfg.OSC.WhelJog_OnlyWhenRun = 0;

			m->pCfg->HeadCfg.OSC.BtnJog_Gain = 4;
			m->pCfg->HeadCfg.OSC.BtnJog_Mode = BTN_JOG_MODE_SINGLE;

			m->pCfg->HeadCfg.OSC.WheelJog_Gain1 = 0.2;
			m->pCfg->HeadCfg.OSC.WhelJog_Mode1 = WHL_JOG_MODE_STEP;

			m->pCfg->HeadCfg.OSC.WheelJog_Gain2 = 0.2;
			m->pCfg->HeadCfg.OSC.WhelJog_Mode2 = WHL_JOG_MODE_STEP;

			m->pCfg->HeadCfg.OSC.DwellDir = 1;

			// WRST
			m->pCfg->HeadCfg.WRST.PROC_Indx = PROC_WRST;
			m->pCfg->HeadCfg.WRST.VECT_A_Indx = VECT_WRST;
			m->pCfg->HeadCfg.WRST.VECT_B_Indx = VECT_WRST;
			m->pCfg->HeadCfg.WRST.TML_A_Indx = TML_AX_WF_1; //TML_AX_WRST;
			m->pCfg->HeadCfg.WRST.TML_B_Indx = TML_AX_WF_1; //TML_AX_WRST;
			m->pCfg->HeadCfg.WRST.Limits_Harcoded = 0;

			m->pCfg->HeadCfg.WRST.BtnJog_Gain = 24.0;
			m->pCfg->HeadCfg.WRST.BtnJog_Mode = BTN_JOG_MODE_SINGLE;

			// AVC
			m->pCfg->HeadCfg.AVC.PROC_Indx = PROC_AVC;
			m->pCfg->HeadCfg.AVC.VECT_A_Indx = VECT_AVC;
			m->pCfg->HeadCfg.AVC.VECT_B_Indx = VECT_AVC2;
			m->pCfg->HeadCfg.AVC.TML_A_Indx = TML_AX_AVC;
			m->pCfg->HeadCfg.AVC.TML_B_Indx = TML_AX_AVC2;

			m->pCfg->HeadCfg.AVC.BtnJog_Gain = 1;
			m->pCfg->HeadCfg.AVC.BtnJog_Mode = BTN_JOG_MODE_SINGLE;

			// GAS
			m->pCfg->HeadCfg.GAS.PROC_Indx = PROC_GAS;

			// COOL
			m->pCfg->HeadCfg.COOL.PROC_Indx = PROC_COOL;

			// TIG
			m->pCfg->HeadCfg.TIG.PROC_Indx = PROC_TIG_PS;

			// HW
			m->pCfg->HeadCfg.HW.PROC_Indx = PROC_HW_PS;

			// INDX
			m->pCfg->HeadCfg.INDX.PROC_Indx = PROC_INDX;
			m->pCfg->HeadCfg.INDX.VECT_A_Indx = VECT_INDX_1;
			m->pCfg->HeadCfg.INDX.VECT_B_Indx = VECT_INDX_2;
			m->pCfg->HeadCfg.INDX.DC_A_Indx = DC_INDX_1;
			m->pCfg->HeadCfg.INDX.DC_B_Indx = DC_INDX_2;
			m->pCfg->HeadCfg.INDX.BtnJog_Gain = 1.0;

			// WB
			m->pCfg->HeadCfg.WB[WB_UD].PROC_Indx = PROC_WB_UD;
			m->pCfg->HeadCfg.WB[WB_LR].PROC_Indx = PROC_WB_LR;

			m->pCfg->HeadCfg.WB[WB_UD].VECT_Indx = VECT_WB_UD;
			m->pCfg->HeadCfg.WB[WB_LR].VECT_Indx = VECT_WB_LR;

			// Lamp On Off
			m->pCfg->HeadCfg.LampOnOFF.VECT_A_Indx = 0; // 0 - not used
			m->pCfg->HeadCfg.LampOnOFF.VECT_B_Indx = 0; // 0 - not used

			/////////////////////////////////////////////////////

			// frame size if zero always speed factor is 1.0
			//m->FrameDia = 4.5 * in_2_mm ;
			m->FrameDia = 0.0;

			Configure_CLAMSHELL_HEAD(m , CLAMSHELL_HEAD);
			DefaultCalibr_CLAMSHELL_HEAD(m->pDefaultCalib);

		break;
		/***************************/
		/***************************/

		/******32 - 33 - 34 ********************/
		case CHERRYPOINT_BP1_HEAD:
		case CHERRYPOINT_BP2_HEAD:
		case CHERRYPOINT_MT_BP2_HEAD:

		// From BPV FLANGE OSC ENC+POT  == BPV_FACE_OSC_EXP

			m->pCfg->HeadCfg.GEN.Torch_Mode = MODE_SINGLE_TORCH;

			// TVL
			m->pCfg->HeadCfg.SwitchHead.VECT_Indx = 0;
			m->pCfg->HeadCfg.SwitchHead.TML_Indx = 0;

			m->pCfg->HeadCfg.TVL.PROC_Indx = PROC_TVL;
			m->pCfg->HeadCfg.TVL.TML_Indx = TML_AX_TVL;

			m->pCfg->HeadCfg.TVL.VECT_Indx = VECT_TVL;
			m->pCfg->HeadCfg.TVL.Enc_Dir = 1;
			//m->pCfg->HeadCfg.TVL.EncPerTick  = 5085;	//	5084.8094458543457034129135792358	// For 1/32 "
			m->pCfg->HeadCfg.TVL.EncPerTick  = 5088; // aby bylo 32 razy
			m->pCfg->HeadCfg.TVL.EncPerTick_SecEnc = 159; // (4000 * 4) / (1" * Pi * 32)
			m->pCfg->HeadCfg.TVL.PinsPerRot = 0;  // Dynamic Configuration
			m->pCfg->HeadCfg.TVL.DistPerTick = 25.4 /32.0; // 1/32"

			m->pCfg->HeadCfg.TVL.BtnJog_Gain = 24;
			m->pCfg->HeadCfg.TVL.BtnJog_Mode = BTN_JOG_MODE_SINGLE;

			// WF
			m->pCfg->HeadCfg.WF.PROC_Indx = PROC_WIRE_FEED;
			m->pCfg->HeadCfg.WF.VECT_A_Indx = VECT_WF;
			m->pCfg->HeadCfg.WF.VECT_B_Indx = VECT_WF_1;
			m->pCfg->HeadCfg.WF.TML_A_Indx = TML_AX_WF;
			m->pCfg->HeadCfg.WF.TML_B_Indx = TML_AX_WF_1;

			m->pCfg->HeadCfg.WF.BtnJog_Gain = 24;
			m->pCfg->HeadCfg.WF.BtnJog_Mode = BTN_JOG_MODE_SINGLE;

			// WP
			m->pCfg->HeadCfg.WP.PROC_Indx = PROC_WIRE_PULSE;
			m->pCfg->HeadCfg.WP.VECT_A_Indx = VECT_WP;
			m->pCfg->HeadCfg.WP.VECT_B_Indx = VECT_WP_1;
			m->pCfg->HeadCfg.WP.TML_A_Indx = TML_AX_WP;
			m->pCfg->HeadCfg.WP.TML_B_Indx = TML_AX_WP_1;

			// OSC
			m->pCfg->HeadCfg.OSC.PROC_Indx = PROC_OSC;
			m->pCfg->HeadCfg.OSC.VECT_A_Indx = VECT_OSC;
			m->pCfg->HeadCfg.OSC.VECT_B_Indx = VECT_OSC;
			m->pCfg->HeadCfg.OSC.TML_A_Indx = TML_AX_OSC;
			m->pCfg->HeadCfg.OSC.TML_B_Indx = TML_AX_OSC;
			m->pCfg->HeadCfg.OSC.Limits_Harcoded = 0;

			m->pCfg->HeadCfg.OSC.WhelJog_OnlyWhenRun = 0;

			m->pCfg->HeadCfg.OSC.BtnJog_Gain = 12;
			m->pCfg->HeadCfg.OSC.BtnJog_Mode = BTN_JOG_MODE_SINGLE;

			m->pCfg->HeadCfg.OSC.WheelJog_Gain1 = 0.2;
			m->pCfg->HeadCfg.OSC.WhelJog_Mode1 = WHL_JOG_MODE_STEP;

			m->pCfg->HeadCfg.OSC.WheelJog_Gain2 = 0.2;
			m->pCfg->HeadCfg.OSC.WhelJog_Mode2 = WHL_JOG_MODE_STEP;

			m->pCfg->HeadCfg.OSC.DwellDir = 1;

			// WRST
			m->pCfg->HeadCfg.WRST.PROC_Indx = PROC_WRST;
			m->pCfg->HeadCfg.WRST.VECT_A_Indx = VECT_WRST;
			m->pCfg->HeadCfg.WRST.VECT_B_Indx = VECT_WRST;
			m->pCfg->HeadCfg.WRST.TML_A_Indx = TML_AX_WRST;
			m->pCfg->HeadCfg.WRST.TML_B_Indx = TML_AX_WRST;
			m->pCfg->HeadCfg.WRST.Limits_Harcoded = 0;

			m->pCfg->HeadCfg.WRST.BtnJog_Gain = 24.0;
			m->pCfg->HeadCfg.WRST.BtnJog_Mode = BTN_JOG_MODE_SINGLE;

			// AVC
			m->pCfg->HeadCfg.AVC.PROC_Indx = PROC_AVC;
			m->pCfg->HeadCfg.AVC.VECT_A_Indx = VECT_AVC;
			m->pCfg->HeadCfg.AVC.VECT_B_Indx = VECT_AVC;
			m->pCfg->HeadCfg.AVC.TML_A_Indx = TML_AX_AVC;
			m->pCfg->HeadCfg.AVC.TML_B_Indx = TML_AX_AVC;

			m->pCfg->HeadCfg.AVC.BtnJog_Gain = 1;
			m->pCfg->HeadCfg.AVC.BtnJog_Mode = BTN_JOG_MODE_SINGLE;

			// GAS
			m->pCfg->HeadCfg.GAS.PROC_Indx = PROC_GAS;

			// COOL
			m->pCfg->HeadCfg.COOL.PROC_Indx = PROC_COOL;

			// TIG
			m->pCfg->HeadCfg.TIG.PROC_Indx = PROC_TIG_PS;

			// HW
			m->pCfg->HeadCfg.HW.PROC_Indx = PROC_HW_PS;

			// INDX
			m->pCfg->HeadCfg.INDX.PROC_Indx = PROC_INDX;
			m->pCfg->HeadCfg.INDX.VECT_A_Indx = VECT_INDX_1;
			m->pCfg->HeadCfg.INDX.VECT_B_Indx = VECT_INDX_2;
			m->pCfg->HeadCfg.INDX.DC_A_Indx = DC_INDX_1;
			m->pCfg->HeadCfg.INDX.DC_B_Indx = DC_INDX_2;
			m->pCfg->HeadCfg.INDX.BtnJog_Gain = 1.0;

			// WB
			m->pCfg->HeadCfg.WB[WB_UD].PROC_Indx = PROC_WB_UD;
			m->pCfg->HeadCfg.WB[WB_LR].PROC_Indx = PROC_WB_LR;

			m->pCfg->HeadCfg.WB[WB_UD].VECT_Indx = VECT_WB_UD;
			m->pCfg->HeadCfg.WB[WB_LR].VECT_Indx = VECT_WB_LR;

			// Lamp On Off
			m->pCfg->HeadCfg.LampOnOFF.VECT_A_Indx = 0; // 0 - not used
			m->pCfg->HeadCfg.LampOnOFF.VECT_B_Indx = 0; // 0 - not used

			/////////////////////////////////////////////////////

			// frame size if zero always speed factor is 1.0
			//m->FrameDia = 4.5 * in_2_mm ;
			m->FrameDia = 0.0;

			switch(headType){

				case CHERRYPOINT_BP1_HEAD:

					Configure_CHERRYPOINT_BPV1_HEAD(m , CHERRYPOINT_BP1_HEAD);
					DefaultCalibr_CHERRYPOINT_BPV1_HEAD(m->pDefaultCalib);

				break;

				case CHERRYPOINT_BP2_HEAD:

					Configure_CHERRYPOINT_BPV2_HEAD(m , CHERRYPOINT_BP2_HEAD);
					DefaultCalibr_CHERRYPOINT_BPV2_HEAD(m->pDefaultCalib);

				break;

				case CHERRYPOINT_MT_BP2_HEAD:

					Configure_CHERRYPOINT_MT_BP2_HEAD(m , CHERRYPOINT_BP2_HEAD);
					DefaultCalibr_CHERRYPOINT_BPV2_HEAD(m->pDefaultCalib);

				break;

			}

		break;

		default:

			// Lamp On Off
			m->pCfg->HeadCfg.LampOnOFF.VECT_A_Indx = 0; // 0 - not used
			m->pCfg->HeadCfg.LampOnOFF.VECT_B_Indx = 0; // 0 - not used

		break;

	}

	PleaseUpdateHeadSetup(m);

	/*********************************************************/
	/****   Parameter assigments   ************************/
	ParametrAssignToPointers( m , 0);

	Process[PROC_TVL].ConfigReady 			= 1;
	Process[PROC_OSC].ConfigReady 			= 1;
	Process[PROC_AVC].ConfigReady 			= 1;
	Process[PROC_WIRE_FEED].ConfigReady 	= 1;
	Process[PROC_WIRE_PULSE].ConfigReady 	= 1;
	Process[PROC_TIG_PS].ConfigReady 		= 1;
	Process[PROC_HW_PS].ConfigReady 		= 1;
	Process[PROC_GAS].ConfigReady 			= 1;
	Process[PROC_COOL].ConfigReady 			= 1;
	Process[PROC_INDX].ConfigReady 			= 1;
	Process[PROC_WRST].ConfigReady 		= 1;
	Process[PROC_WB_UD].ConfigReady 		= 1;
	Process[PROC_WB_LR].ConfigReady 		= 1;
```
